Yaskawa INFORM job: u_tourne3TRJ4.JBI

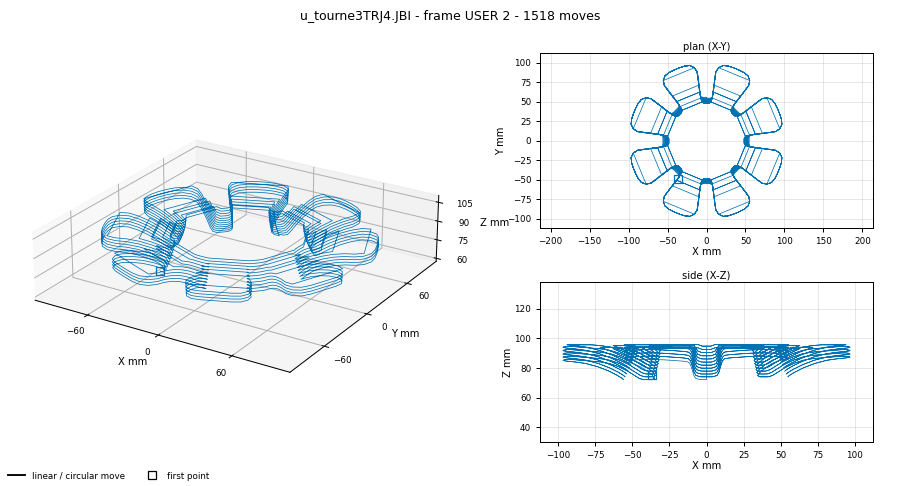
[picture p0: tool path of u_tourne3TRJ4.JBI in frame USER 2, 1518 of 1518 moves have a stored position in this frame; points joined in program order, loops and branches not executed]
/JOB
//NAME u_tourne3TRJ4
///FOLDERNAME DEMO
//POS
///NPOS 1518,0,1518,0,0,0
///USER 2
///TOOL 7
///POSTYPE USER
///RECTAN
///RCONF 1,0,0,0,0,0,0,0,0,0,0,0,0,0,0,0,0,0,0,0,0,0,0,0
C00000=-36.517,-48.718,75.143,177.9288,-0.0843,-14346.8537
C00001=-35.037,-45.351,73.015,-166.0442,10.7217,-14347.6887
C00002=-36.538,-42.505,72.166,-173.7278,29.8093,-14350.6829
C00003=-38.303,-40.803,72.129,179.7748,31.2094,-14353.1899
C00004=-39.567,-39.567,72.154,-180.0000,31.1989,-14355.0000
C00005=-40.803,-38.303,72.129,-179.7748,31.2094,-14356.8101
C00006=-42.506,-36.538,72.166,173.7274,29.8092,-14359.3178
C00007=-45.352,-35.037,73.015,166.0441,10.7215,-14362.3119
C00008=-48.718,-36.517,75.143,-177.9288,-0.0843,-14363.1463
C00009=-53.324,-40.007,78.036,-176.1608,-0.0420,-14363.1205
C00010=-59.196,-44.618,80.927,-175.6070,-0.0220,-14362.9934
C00011=-65.578,-49.604,83.062,-175.3163,-0.0261,-14362.8957
C00012=-71.524,-53.949,84.088,-175.5865,-0.7799,-14362.9735
C00013=-77.795,-55.184,84.621,-177.8577,-1.8362,-14364.6500
C00014=-83.601,-53.037,85.050,-179.4963,-1.2492,-14367.6087
C00015=-87.741,-47.957,85.481,179.9995,-0.0846,-14371.3401
C00016=-90.934,-41.602,85.762,-179.9996,-0.0128,-14375.4161
C00017=-93.717,-34.883,85.762,-179.9986,-0.0127,-14379.5839
C00018=-95.953,-28.131,85.481,179.9978,-0.0889,-14383.6602
C00019=-96.617,-21.612,85.050,179.4972,-1.2499,-14387.3912
C00020=-94.030,-15.989,84.621,177.8561,-1.8342,-14390.3496
C00021=-88.723,-12.427,84.088,175.5876,-0.7793,-14392.0267
C00022=-81.446,-11.295,83.062,175.3181,-0.0225,-14392.1045
C00023=-73.408,-10.308,80.927,175.6017,-0.0195,-14392.0068
C00024=-65.995,-9.417,78.036,176.1598,-0.0428,-14391.8791
C00025=-60.270,-8.627,75.143,177.9267,-0.0854,-14391.8541
C00026=-56.844,-7.293,73.015,-166.0480,10.7254,-14392.6890
C00027=-55.892,-4.219,72.166,-173.7293,29.8078,-14395.6832
C00028=-55.936,-1.768,72.129,179.7768,31.2086,-14398.1896
C00029=-55.957,0.000,72.154,-180.0000,31.1976,-14400.0000
C00030=-55.936,1.767,72.129,-179.7762,31.2086,-14401.8094
C00031=-55.892,4.220,72.166,173.7222,29.8074,-14404.3178
C00032=-56.844,7.293,73.015,166.0480,10.7254,-14407.3110
C00033=-60.270,8.627,75.143,-177.9267,-0.0854,-14408.1459
C00034=-65.995,9.417,78.036,-176.1598,-0.0428,-14408.1209
C00035=-73.408,10.308,80.927,-175.6017,-0.0195,-14407.9932
C00036=-81.446,11.295,83.062,-175.3181,-0.0225,-14407.8955
C00037=-88.723,12.427,84.088,-175.5876,-0.7793,-14407.9733
C00038=-94.030,15.989,84.621,-177.8561,-1.8342,-14409.6504
C00039=-96.617,21.612,85.050,-179.4972,-1.2499,-14412.6088
C00040=-95.953,28.131,85.481,-179.9978,-0.0889,-14416.3398
C00041=-93.717,34.883,85.762,179.9986,-0.0127,-14420.4161
C00042=-90.934,41.602,85.762,179.9996,-0.0128,-14424.5839
C00043=-87.741,47.957,85.481,-179.9995,-0.0846,-14428.6599
C00044=-83.601,53.037,85.050,179.4963,-1.2492,-14432.3913
C00045=-77.795,55.184,84.621,177.8577,-1.8362,-14435.3500
C00046=-71.524,53.949,84.088,175.5865,-0.7799,-14437.0265
C00047=-65.578,49.604,83.062,175.3163,-0.0261,-14437.1043
C00048=-59.196,44.618,80.927,175.6070,-0.0220,-14437.0066
C00049=-53.324,40.007,78.036,176.1608,-0.0420,-14436.8795
C00050=-48.718,36.517,75.143,177.9288,-0.0843,-14436.8537
C00051=-45.351,35.037,73.015,-166.0442,10.7217,-14437.6887
C00052=-42.505,36.538,72.166,-173.7278,29.8093,-14440.6829
C00053=-40.803,38.303,72.129,179.7748,31.2094,-14443.1899
C00054=-39.567,39.567,72.154,-180.0000,31.1989,-14445.0000
C00055=-38.303,40.803,72.129,-179.7748,31.2094,-14446.8101
C00056=-36.538,42.506,72.166,173.7274,29.8092,-14449.3178
C00057=-35.037,45.352,73.015,166.0441,10.7215,-14452.3119
C00058=-36.517,48.718,75.143,-177.9288,-0.0843,-14453.1463
C00059=-40.007,53.324,78.036,-176.1608,-0.0420,-14453.1205
C00060=-44.618,59.196,80.927,-175.6070,-0.0220,-14452.9934
C00061=-49.604,65.578,83.062,-175.3163,-0.0261,-14452.8957
C00062=-53.949,71.524,84.088,-175.5865,-0.7799,-14452.9735
C00063=-55.184,77.795,84.621,-177.8577,-1.8362,-14454.6500
C00064=-53.037,83.601,85.050,-179.4963,-1.2492,-14457.6087
C00065=-47.957,87.741,85.481,179.9995,-0.0846,-14461.3401
C00066=-41.602,90.934,85.762,-179.9996,-0.0128,-14465.4161
C00067=-34.883,93.717,85.762,-179.9986,-0.0127,-14469.5839
C00068=-28.131,95.953,85.481,179.9978,-0.0889,-14473.6602
C00069=-21.612,96.617,85.050,179.4972,-1.2499,-14477.3912
C00070=-15.989,94.030,84.621,177.8561,-1.8342,-14480.3496
C00071=-12.427,88.723,84.088,175.5876,-0.7793,-14482.0267
C00072=-11.295,81.446,83.062,175.3181,-0.0225,-14482.1045
C00073=-10.308,73.408,80.927,175.6017,-0.0195,-14482.0068
C00074=-9.417,65.995,78.036,176.1598,-0.0428,-14481.8791
C00075=-8.627,60.270,75.143,177.9267,-0.0854,-14481.8541
C00076=-7.293,56.844,73.015,-166.0480,10.7254,-14482.6890
C00077=-4.220,55.892,72.166,-173.7222,29.8074,-14485.6822
C00078=-1.767,55.936,72.129,179.7762,31.2086,-14488.1906
C00079=0.000,55.957,72.154,-180.0000,31.1976,-14490.0000
C00080=0.000,54.840,74.049,-180.0000,29.7413,-14490.0000
C00081=1.666,54.823,74.024,-179.8067,29.7500,-14491.7406
C00082=4.048,54.790,74.062,173.8586,28.2915,-14494.2255
C00083=7.088,55.804,74.943,167.0788,9.5543,-14497.2387
C00084=8.393,59.388,77.145,-177.8370,-0.0706,-14498.0440
C00085=9.180,65.335,80.122,-176.4294,-0.0310,-14497.9981
C00086=10.089,72.980,83.074,-176.0907,-0.0153,-14497.8709
C00087=11.094,81.206,85.240,-175.9759,-0.0117,-14497.7793
C00088=12.226,88.613,86.276,-176.2817,-0.6456,-14497.8555
C00089=15.808,94.009,86.813,-178.2035,-1.5233,-14499.5452
C00090=21.475,96.642,87.246,-179.5823,-1.0342,-14502.5282
C00091=28.048,95.980,87.679,179.9973,-0.0724,-14506.2898
C00092=34.856,93.728,87.962,179.9966,-0.0074,-14510.3994
C00093=41.629,90.922,87.962,179.9972,-0.0076,-14514.6009
C00094=48.035,87.701,87.679,-179.9999,-0.0718,-14518.7101
C00095=53.151,83.521,87.246,179.5838,-1.0323,-14522.4718
C00096=55.296,77.652,86.813,178.2066,-1.5235,-14525.4547
C00097=54.014,71.304,86.276,176.2804,-0.6460,-14527.1446
C00098=49.577,65.266,85.240,175.9790,-0.0155,-14527.2208
C00099=44.470,58.738,83.074,176.0895,-0.0120,-14527.1290
C00100=39.708,52.690,80.122,176.4261,-0.0301,-14527.0022
C00101=36.059,47.928,77.145,177.8373,-0.0709,-14526.9563
C00102=34.447,44.472,74.943,-167.0757,9.5522,-14527.7605
C00103=35.880,41.605,74.062,-173.8568,28.2919,-14530.7744
C00104=37.588,39.944,74.024,179.8046,29.7498,-14533.2595
C00105=38.778,38.778,74.049,-180.0000,29.7416,-14535.0000
C00106=39.943,37.588,74.024,-179.8042,29.7498,-14536.7398
C00107=41.605,35.880,74.062,173.8533,28.2853,-14539.2256
C00108=44.472,34.447,74.943,167.0757,9.5522,-14542.2395
C00109=47.928,36.059,77.145,-177.8373,-0.0709,-14543.0437
C00110=52.690,39.708,80.122,-176.4261,-0.0301,-14542.9978
C00111=58.738,44.470,83.074,-176.0895,-0.0120,-14542.8710
C00112=65.266,49.577,85.240,-175.9790,-0.0155,-14542.7792
C00113=71.304,54.014,86.276,-176.2804,-0.6460,-14542.8554
C00114=77.652,55.296,86.813,-178.2066,-1.5235,-14544.5453
C00115=83.521,53.151,87.246,-179.5838,-1.0323,-14547.5282
C00116=87.701,48.035,87.679,179.9999,-0.0718,-14551.2899
C00117=90.922,41.629,87.962,-179.9972,-0.0076,-14555.3991
C00118=93.728,34.856,87.962,-179.9966,-0.0074,-14559.6006
C00119=95.980,28.048,87.679,-179.9973,-0.0724,-14563.7102
C00120=96.642,21.475,87.246,179.5823,-1.0342,-14567.4718
C00121=94.009,15.808,86.813,178.2035,-1.5233,-14570.4548
C00122=88.613,12.226,86.276,176.2817,-0.6456,-14572.1445
C00123=81.206,11.094,85.240,175.9759,-0.0117,-14572.2207
C00124=72.980,10.089,83.074,176.0907,-0.0153,-14572.1291
C00125=65.335,9.180,80.122,176.4294,-0.0310,-14572.0019
C00126=59.388,8.393,77.145,177.8370,-0.0706,-14571.9560
C00127=55.804,7.088,74.943,-167.0788,9.5543,-14572.7613
C00128=54.790,4.048,74.062,-173.8586,28.2915,-14575.7745
C00129=54.823,1.666,74.024,179.8067,29.7500,-14578.2594
C00130=54.840,0.000,74.049,180.0000,29.7413,-14580.0000
C00131=54.823,-1.665,74.024,-179.8061,29.7500,-14581.7396
C00132=54.790,-4.048,74.062,173.8593,28.2888,-14584.2255
C00133=55.804,-7.088,74.943,167.0788,9.5543,-14587.2387
C00134=59.388,-8.393,77.145,-177.8370,-0.0706,-14588.0440
C00135=65.335,-9.180,80.122,-176.4294,-0.0310,-14587.9981
C00136=72.980,-10.089,83.074,-176.0907,-0.0153,-14587.8709
C00137=81.206,-11.094,85.240,-175.9759,-0.0117,-14587.7793
C00138=88.613,-12.226,86.276,-176.2817,-0.6456,-14587.8555
C00139=94.009,-15.808,86.813,-178.2035,-1.5233,-14589.5452
C00140=96.642,-21.475,87.246,-179.5823,-1.0342,-14592.5282
C00141=95.980,-28.048,87.679,179.9973,-0.0724,-14596.2898
C00142=93.728,-34.856,87.962,179.9966,-0.0074,-14600.3994
C00143=90.922,-41.629,87.962,179.9972,-0.0076,-14604.6009
C00144=87.701,-48.035,87.679,-179.9999,-0.0718,-14608.7101
C00145=83.521,-53.151,87.246,179.5838,-1.0323,-14612.4718
C00146=77.652,-55.296,86.813,178.2066,-1.5235,-14615.4547
C00147=71.304,-54.014,86.276,176.2804,-0.6460,-14617.1446
C00148=65.266,-49.577,85.240,175.9790,-0.0155,-14617.2208
C00149=58.738,-44.470,83.074,176.0895,-0.0120,-14617.1290
C00150=52.690,-39.708,80.122,176.4261,-0.0301,-14617.0022
C00151=47.928,-36.059,77.145,177.8373,-0.0709,-14616.9563
C00152=44.472,-34.447,74.943,-167.0757,9.5522,-14617.7605
C00153=41.605,-35.880,74.062,-173.8568,28.2919,-14620.7744
C00154=39.944,-37.588,74.024,179.8046,29.7498,-14623.2595
C00155=38.778,-38.778,74.049,180.0000,29.7416,-14625.0000
C00156=37.588,-39.943,74.024,-179.8042,29.7498,-14626.7398
C00157=35.880,-41.605,74.062,173.8533,28.2853,-14629.2256
C00158=34.447,-44.472,74.943,167.0757,9.5522,-14632.2395
C00159=36.059,-47.928,77.145,-177.8373,-0.0709,-14633.0437
C00160=39.708,-52.690,80.122,-176.4261,-0.0301,-14632.9978
C00161=44.470,-58.738,83.074,-176.0895,-0.0120,-14632.8710
C00162=49.577,-65.266,85.240,-175.9790,-0.0155,-14632.7792
C00163=54.014,-71.304,86.276,-176.2804,-0.6460,-14632.8554
C00164=55.296,-77.652,86.813,-178.2066,-1.5235,-14634.5453
C00165=53.151,-83.521,87.246,-179.5838,-1.0323,-14637.5282
C00166=48.035,-87.701,87.679,179.9999,-0.0718,-14641.2899
C00167=41.629,-90.922,87.962,-179.9972,-0.0076,-14645.3991
C00168=34.856,-93.728,87.962,-179.9966,-0.0074,-14649.6006
C00169=28.048,-95.980,87.679,-179.9973,-0.0724,-14653.7102
C00170=21.475,-96.642,87.246,179.5823,-1.0342,-14657.4718
C00171=15.808,-94.009,86.813,178.2035,-1.5233,-14660.4548
C00172=12.226,-88.613,86.276,176.2817,-0.6456,-14662.1445
C00173=11.094,-81.206,85.240,175.9759,-0.0117,-14662.2207
C00174=10.089,-72.980,83.074,176.0907,-0.0153,-14662.1291
C00175=9.180,-65.335,80.122,176.4294,-0.0310,-14662.0019
C00176=8.393,-59.388,77.145,177.8370,-0.0706,-14661.9560
C00177=7.088,-55.804,74.943,-167.0788,9.5543,-14662.7613
C00178=4.048,-54.790,74.062,-173.8586,28.2915,-14665.7745
C00179=1.666,-54.823,74.024,179.8067,29.7500,-14668.2594
C00180=0.000,-54.840,74.049,-180.0000,29.7413,-14670.0000
C00181=0.000,-54.840,74.049,-180.0000,29.7413,-14670.0000
C00182=-1.665,-54.823,74.024,-179.8061,29.7500,-14671.7396
C00183=-4.048,-54.790,74.062,173.8593,28.2888,-14674.2255
C00184=-7.088,-55.804,74.943,167.0788,9.5543,-14677.2387
C00185=-8.393,-59.388,77.145,-177.8370,-0.0706,-14678.0440
C00186=-9.180,-65.335,80.122,-176.4294,-0.0310,-14677.9981
C00187=-10.089,-72.980,83.074,-176.0907,-0.0153,-14677.8709
C00188=-11.094,-81.206,85.240,-175.9759,-0.0117,-14677.7793
C00189=-12.226,-88.613,86.276,-176.2817,-0.6456,-14677.8555
C00190=-15.808,-94.009,86.813,-178.2035,-1.5233,-14679.5452
C00191=-21.475,-96.642,87.246,-179.5823,-1.0342,-14682.5282
C00192=-28.048,-95.980,87.679,179.9973,-0.0724,-14686.2898
C00193=-34.856,-93.728,87.962,179.9966,-0.0074,-14690.3994
C00194=-41.629,-90.922,87.962,179.9972,-0.0076,-14694.6009
C00195=-48.035,-87.701,87.679,-179.9999,-0.0718,-14698.7101
C00196=-53.151,-83.521,87.246,179.5838,-1.0323,-14702.4718
C00197=-55.296,-77.652,86.813,178.2066,-1.5235,-14705.4547
C00198=-54.014,-71.304,86.276,176.2804,-0.6460,-14707.1446
C00199=-49.577,-65.266,85.240,175.9790,-0.0155,-14707.2208
C00200=-44.470,-58.738,83.074,176.0895,-0.0120,-14707.1290
C00201=-39.708,-52.690,80.122,176.4261,-0.0301,-14707.0022
C00202=-36.059,-47.928,77.145,177.8373,-0.0709,-14706.9563
C00203=-34.447,-44.472,74.943,-167.0757,9.5522,-14707.7605
C00204=-35.880,-41.605,74.062,-173.8568,28.2919,-14710.7744
C00205=-37.588,-39.944,74.024,179.8046,29.7498,-14713.2595
C00206=-38.778,-38.778,74.049,-180.0000,29.7416,-14715.0000
C00207=-39.943,-37.588,74.024,-179.8042,29.7498,-14716.7398
C00208=-41.605,-35.880,74.062,173.8533,28.2853,-14719.2256
C00209=-44.472,-34.447,74.943,167.0757,9.5522,-14722.2395
C00210=-47.928,-36.059,77.145,-177.8373,-0.0709,-14723.0437
C00211=-52.690,-39.708,80.122,-176.4261,-0.0301,-14722.9978
C00212=-58.738,-44.470,83.074,-176.0895,-0.0120,-14722.8710
C00213=-65.266,-49.577,85.240,-175.9790,-0.0155,-14722.7792
C00214=-71.304,-54.014,86.276,-176.2804,-0.6460,-14722.8554
C00215=-77.652,-55.296,86.813,-178.2066,-1.5235,-14724.5453
C00216=-83.521,-53.151,87.246,-179.5838,-1.0323,-14727.5282
C00217=-87.701,-48.035,87.679,179.9999,-0.0718,-14731.2899
C00218=-90.922,-41.629,87.962,-179.9972,-0.0076,-14735.3991
C00219=-93.728,-34.856,87.962,-179.9966,-0.0074,-14739.6006
C00220=-95.980,-28.048,87.679,-179.9973,-0.0724,-14743.7102
C00221=-96.642,-21.475,87.246,179.5823,-1.0342,-14747.4718
C00222=-94.009,-15.808,86.813,178.2035,-1.5233,-14750.4548
C00223=-88.613,-12.226,86.276,176.2817,-0.6456,-14752.1445
C00224=-81.206,-11.094,85.240,175.9759,-0.0117,-14752.2207
C00225=-72.980,-10.089,83.074,176.0907,-0.0153,-14752.1291
C00226=-65.335,-9.180,80.122,176.4294,-0.0310,-14752.0019
C00227=-59.388,-8.393,77.145,177.8370,-0.0706,-14751.9560
C00228=-55.804,-7.088,74.943,-167.0788,9.5543,-14752.7613
C00229=-54.790,-4.048,74.062,-173.8586,28.2915,-14755.7745
C00230=-54.823,-1.666,74.024,179.8067,29.7500,-14758.2594
C00231=-54.840,0.000,74.049,-180.0000,29.7413,-14760.0000
C00232=-54.823,1.665,74.024,-179.8061,29.7500,-14761.7396
C00233=-54.790,4.048,74.062,173.8593,28.2888,-14764.2255
C00234=-55.804,7.088,74.943,167.0788,9.5543,-14767.2387
C00235=-59.388,8.393,77.145,-177.8370,-0.0706,-14768.0440
C00236=-65.335,9.180,80.122,-176.4294,-0.0310,-14767.9981
C00237=-72.980,10.089,83.074,-176.0907,-0.0153,-14767.8709
C00238=-81.206,11.094,85.240,-175.9759,-0.0117,-14767.7793
C00239=-88.613,12.226,86.276,-176.2817,-0.6456,-14767.8555
C00240=-94.009,15.808,86.813,-178.2035,-1.5233,-14769.5452
C00241=-96.642,21.475,87.246,-179.5823,-1.0342,-14772.5282
C00242=-95.980,28.048,87.679,179.9973,-0.0724,-14776.2898
C00243=-93.728,34.856,87.962,179.9966,-0.0074,-14780.3994
C00244=-90.922,41.629,87.962,179.9972,-0.0076,-14784.6009
C00245=-87.701,48.035,87.679,-179.9999,-0.0718,-14788.7101
C00246=-83.521,53.151,87.246,179.5838,-1.0323,-14792.4718
C00247=-77.652,55.296,86.813,178.2066,-1.5235,-14795.4547
C00248=-71.304,54.014,86.276,176.2804,-0.6460,-14797.1446
C00249=-65.266,49.577,85.240,175.9790,-0.0155,-14797.2208
C00250=-58.738,44.470,83.074,176.0895,-0.0120,-14797.1290
C00251=-52.690,39.708,80.122,176.4261,-0.0301,-14797.0022
C00252=-47.928,36.059,77.145,177.8373,-0.0709,-14796.9563
C00253=-44.472,34.447,74.943,-167.0757,9.5522,-14797.7605
C00254=-41.605,35.880,74.062,-173.8568,28.2919,-14800.7744
C00255=-39.944,37.588,74.024,179.8046,29.7498,-14803.2595
C00256=-38.778,38.778,74.049,-180.0000,29.7416,-14805.0000
C00257=-37.588,39.943,74.024,-179.8042,29.7498,-14806.7398
C00258=-35.880,41.605,74.062,173.8533,28.2853,-14809.2256
C00259=-34.447,44.472,74.943,167.0757,9.5522,-14812.2395
C00260=-36.059,47.928,77.145,-177.8373,-0.0709,-14813.0437
C00261=-39.708,52.690,80.122,-176.4261,-0.0301,-14812.9978
C00262=-44.470,58.738,83.074,-176.0895,-0.0120,-14812.8710
C00263=-49.577,65.266,85.240,-175.9790,-0.0155,-14812.7792
C00264=-54.014,71.304,86.276,-176.2804,-0.6460,-14812.8554
C00265=-55.296,77.652,86.813,-178.2066,-1.5235,-14814.5453
C00266=-53.151,83.521,87.246,-179.5838,-1.0323,-14817.5282
C00267=-48.035,87.701,87.679,179.9999,-0.0718,-14821.2899
C00268=-41.629,90.922,87.962,-179.9972,-0.0076,-14825.3991
C00269=-34.856,93.728,87.962,-179.9966,-0.0074,-14829.6006
C00270=-28.048,95.980,87.679,-179.9973,-0.0724,-14833.7102
C00271=-21.475,96.642,87.246,179.5823,-1.0342,-14837.4718
C00272=-15.808,94.009,86.813,178.2035,-1.5233,-14840.4548
C00273=-12.226,88.613,86.276,176.2817,-0.6456,-14842.1445
C00274=-11.094,81.206,85.240,175.9759,-0.0117,-14842.2207
C00275=-10.089,72.980,83.074,176.0907,-0.0153,-14842.1291
C00276=-9.180,65.335,80.122,176.4294,-0.0310,-14842.0019
C00277=-8.393,59.388,77.145,177.8370,-0.0706,-14841.9560
C00278=-7.088,55.804,74.943,-167.0788,9.5543,-14842.7613
C00279=-4.048,54.790,74.062,-173.8593,28.2888,-14845.7745
C00280=-1.665,54.823,74.024,179.8061,29.7500,-14848.2604
C00281=0.000,54.840,74.049,180.0000,29.7413,-14850.0000
C00282=0.000,53.776,75.975,180.0000,28.1001,-14850.0000
C00283=1.568,53.762,75.948,-179.8334,28.1117,-14851.6706
C00284=3.884,53.739,75.988,174.0567,26.6026,-14854.1339
C00285=6.894,54.818,76.900,168.1623,8.4382,-14857.1680
C00286=8.175,58.565,79.173,-177.8225,-0.0548,-14857.9465
C00287=8.965,64.737,82.228,-176.7507,-0.0188,-14857.8844
C00288=9.898,72.606,85.234,-176.6314,-0.0094,-14857.7630
C00289=10.924,81.005,87.424,-176.6961,-0.0057,-14857.6803
C00290=12.061,88.524,88.468,-177.0328,-0.5045,-14857.7585
C00291=15.662,93.991,89.008,-178.5867,-1.1939,-14859.4604
C00292=21.365,96.662,89.443,-179.6771,-0.7971,-14862.4636
C00293=27.983,96.002,89.878,179.9979,-0.0543,-14866.2505
C00294=34.834,93.736,90.162,-179.9980,-0.0054,-14870.3860
C00295=41.650,90.913,90.162,-179.9976,-0.0052,-14874.6140
C00296=48.097,87.670,89.878,179.9969,-0.0540,-14878.7498
C00297=53.243,83.458,89.443,179.6739,-0.7993,-14882.5363
C00298=55.387,77.537,89.008,178.5849,-1.1940,-14885.5394
C00299=54.067,71.124,88.468,177.0304,-0.5081,-14887.2413
C00300=49.554,65.004,87.424,176.6978,-0.0087,-14887.3191
C00301=44.341,58.339,85.234,176.6315,-0.0113,-14887.2369
C00302=39.437,52.115,82.228,176.7520,-0.0208,-14887.1159
C00303=35.631,47.192,79.173,177.8236,-0.0563,-14887.0536
C00304=33.888,43.637,76.900,-168.1624,8.4405,-14887.8325
C00305=35.253,40.746,75.988,-174.0559,26.5997,-14890.8660
C00306=36.906,39.124,75.948,179.8313,28.1098,-14893.3290
C00307=38.025,38.025,75.975,-180.0000,28.0967,-14895.0000
C00308=39.124,36.906,75.948,-179.8313,28.1098,-14896.6710
C00309=40.746,35.253,75.988,174.0559,26.5997,-14899.1340
C00310=43.637,33.888,76.901,168.1624,8.4405,-14902.1675
C00311=47.192,35.631,79.173,-177.8236,-0.0563,-14902.9464
C00312=52.115,39.437,82.228,-176.7520,-0.0208,-14902.8841
C00313=58.339,44.341,85.234,-176.6315,-0.0113,-14902.7631
C00314=65.004,49.554,87.424,-176.6978,-0.0087,-14902.6809
C00315=71.124,54.067,88.468,-177.0304,-0.5081,-14902.7587
C00316=77.537,55.387,89.008,-178.5849,-1.1940,-14904.4606
C00317=83.458,53.243,89.443,-179.6739,-0.7993,-14907.4637
C00318=87.670,48.097,89.878,-179.9969,-0.0540,-14911.2502
C00319=90.913,41.650,90.162,179.9976,-0.0052,-14915.3860
C00320=93.736,34.834,90.162,179.9980,-0.0054,-14919.6140
C00321=96.002,27.983,89.878,-179.9979,-0.0543,-14923.7495
C00322=96.662,21.365,89.443,179.6771,-0.7971,-14927.5364
C00323=93.991,15.662,89.008,178.5867,-1.1939,-14930.5396
C00324=88.524,12.061,88.468,177.0328,-0.5045,-14932.2415
C00325=81.005,10.924,87.424,176.6961,-0.0057,-14932.3197
C00326=72.606,9.898,85.234,176.6314,-0.0094,-14932.2370
C00327=64.737,8.965,82.228,176.7507,-0.0188,-14932.1156
C00328=58.565,8.175,79.173,177.8225,-0.0548,-14932.0535
C00329=54.818,6.894,76.900,-168.1623,8.4382,-14932.8320
C00330=53.739,3.884,75.988,-174.0567,26.6026,-14935.8661
C00331=53.762,1.568,75.948,179.8334,28.1117,-14938.3294
C00332=53.776,0.000,75.975,180.0000,28.1001,-14940.0000
C00333=53.762,-1.568,75.948,-179.8334,28.1117,-14941.6706
C00334=53.739,-3.885,75.988,174.0562,26.6025,-14944.1349
C00335=54.819,-6.894,76.901,168.1623,8.4383,-14947.1678
C00336=58.565,-8.175,79.173,-177.8225,-0.0548,-14947.9465
C00337=64.737,-8.965,82.228,-176.7507,-0.0188,-14947.8844
C00338=72.606,-9.898,85.234,-176.6314,-0.0094,-14947.7630
C00339=81.005,-10.924,87.424,-176.6961,-0.0057,-14947.6803
C00340=88.524,-12.061,88.468,-177.0328,-0.5045,-14947.7585
C00341=93.991,-15.662,89.008,-178.5867,-1.1939,-14949.4604
C00342=96.662,-21.365,89.443,-179.6771,-0.7971,-14952.4636
C00343=96.002,-27.983,89.878,179.9979,-0.0543,-14956.2505
C00344=93.736,-34.834,90.162,-179.9980,-0.0054,-14960.3860
C00345=90.913,-41.650,90.162,-179.9976,-0.0052,-14964.6140
C00346=87.670,-48.097,89.878,179.9969,-0.0540,-14968.7498
C00347=83.458,-53.243,89.443,179.6739,-0.7993,-14972.5363
C00348=77.537,-55.387,89.008,178.5849,-1.1940,-14975.5394
C00349=71.124,-54.067,88.468,177.0304,-0.5081,-14977.2413
C00350=65.004,-49.554,87.424,176.6978,-0.0087,-14977.3191
C00351=58.339,-44.341,85.234,176.6315,-0.0113,-14977.2369
C00352=52.115,-39.437,82.228,176.7520,-0.0208,-14977.1159
C00353=47.192,-35.631,79.173,177.8236,-0.0563,-14977.0536
C00354=43.637,-33.888,76.900,-168.1624,8.4405,-14977.8325
C00355=40.746,-35.253,75.988,-174.0559,26.5997,-14980.8660
C00356=39.124,-36.906,75.948,179.8313,28.1098,-14983.3290
C00357=38.025,-38.025,75.975,-180.0000,28.0967,-14985.0000
C00358=36.906,-39.124,75.948,-179.8313,28.1098,-14986.6710
C00359=35.253,-40.746,75.988,174.0559,26.5997,-14989.1340
C00360=33.888,-43.637,76.901,168.1624,8.4405,-14992.1675
C00361=35.631,-47.192,79.173,-177.8236,-0.0563,-14992.9464
C00362=39.437,-52.115,82.228,-176.7520,-0.0208,-14992.8841
C00363=44.341,-58.339,85.234,-176.6315,-0.0113,-14992.7631
C00364=49.554,-65.004,87.424,-176.6978,-0.0087,-14992.6809
C00365=54.067,-71.124,88.468,-177.0304,-0.5081,-14992.7587
C00366=55.387,-77.537,89.008,-178.5849,-1.1940,-14994.4606
C00367=53.243,-83.458,89.443,-179.6739,-0.7993,-14997.4637
C00368=48.097,-87.670,89.878,-179.9969,-0.0540,-15001.2502
C00369=41.650,-90.913,90.162,179.9976,-0.0052,-15005.3860
C00370=34.834,-93.736,90.162,179.9980,-0.0054,-15009.6140
C00371=27.983,-96.002,89.878,-179.9979,-0.0543,-15013.7495
C00372=21.365,-96.662,89.443,179.6771,-0.7971,-15017.5364
C00373=15.662,-93.991,89.008,178.5867,-1.1939,-15020.5396
C00374=12.061,-88.524,88.468,177.0328,-0.5045,-15022.2415
C00375=10.924,-81.005,87.424,176.6961,-0.0057,-15022.3197
C00376=9.898,-72.606,85.234,176.6314,-0.0094,-15022.2370
C00377=8.965,-64.737,82.228,176.7507,-0.0188,-15022.1156
C00378=8.175,-58.565,79.173,177.8225,-0.0548,-15022.0535
C00379=6.894,-54.818,76.900,-168.1623,8.4382,-15022.8320
C00380=3.884,-53.739,75.988,-174.0567,26.6026,-15025.8661
C00381=1.568,-53.762,75.948,179.8334,28.1117,-15028.3294
C00382=0.000,-53.776,75.975,180.0000,28.1001,-15030.0000
C00383=0.000,-53.776,75.975,180.0000,28.1001,-15030.0000
C00384=-1.568,-53.762,75.948,-179.8334,28.1117,-15031.6706
C00385=-3.885,-53.739,75.988,174.0562,26.6025,-15034.1349
C00386=-6.894,-54.819,76.901,168.1623,8.4383,-15037.1678
C00387=-8.175,-58.565,79.173,-177.8225,-0.0548,-15037.9465
C00388=-8.965,-64.737,82.228,-176.7507,-0.0188,-15037.8844
C00389=-9.898,-72.606,85.234,-176.6314,-0.0094,-15037.7630
C00390=-10.924,-81.005,87.424,-176.6961,-0.0057,-15037.6803
C00391=-12.061,-88.524,88.468,-177.0328,-0.5045,-15037.7585
C00392=-15.662,-93.991,89.008,-178.5867,-1.1939,-15039.4604
C00393=-21.365,-96.662,89.443,-179.6771,-0.7971,-15042.4636
C00394=-27.983,-96.002,89.878,179.9979,-0.0543,-15046.2505
C00395=-34.834,-93.736,90.162,-179.9980,-0.0054,-15050.3860
C00396=-41.650,-90.913,90.162,-179.9976,-0.0052,-15054.6140
C00397=-48.097,-87.670,89.878,179.9969,-0.0540,-15058.7498
C00398=-53.243,-83.458,89.443,179.6739,-0.7993,-15062.5363
C00399=-55.387,-77.537,89.008,178.5849,-1.1940,-15065.5394
C00400=-54.067,-71.124,88.468,177.0304,-0.5081,-15067.2413
C00401=-49.554,-65.004,87.424,176.6978,-0.0087,-15067.3191
C00402=-44.341,-58.339,85.234,176.6315,-0.0113,-15067.2369
C00403=-39.437,-52.115,82.228,176.7520,-0.0208,-15067.1159
C00404=-35.631,-47.192,79.173,177.8236,-0.0563,-15067.0536
C00405=-33.888,-43.637,76.900,-168.1624,8.4405,-15067.8325
C00406=-35.253,-40.746,75.988,-174.0559,26.5997,-15070.8660
C00407=-36.906,-39.124,75.948,179.8313,28.1098,-15073.3290
C00408=-38.025,-38.025,75.975,-180.0000,28.0967,-15075.0000
C00409=-39.124,-36.906,75.948,-179.8313,28.1098,-15076.6710
C00410=-40.746,-35.253,75.988,174.0559,26.5997,-15079.1340
C00411=-43.637,-33.888,76.901,168.1624,8.4405,-15082.1675
C00412=-47.192,-35.631,79.173,-177.8236,-0.0563,-15082.9464
C00413=-52.115,-39.437,82.228,-176.7520,-0.0208,-15082.8841
C00414=-58.339,-44.341,85.234,-176.6315,-0.0113,-15082.7631
C00415=-65.004,-49.554,87.424,-176.6978,-0.0087,-15082.6809
C00416=-71.124,-54.067,88.468,-177.0304,-0.5081,-15082.7587
C00417=-77.537,-55.387,89.008,-178.5849,-1.1940,-15084.4606
C00418=-83.458,-53.243,89.443,-179.6739,-0.7993,-15087.4637
C00419=-87.670,-48.097,89.878,-179.9969,-0.0540,-15091.2502
C00420=-90.913,-41.650,90.162,179.9976,-0.0052,-15095.3860
C00421=-93.736,-34.834,90.162,179.9980,-0.0054,-15099.6140
C00422=-96.002,-27.983,89.878,-179.9979,-0.0543,-15103.7495
C00423=-96.662,-21.365,89.443,179.6771,-0.7971,-15107.5364
C00424=-93.991,-15.662,89.008,178.5867,-1.1939,-15110.5396
C00425=-88.524,-12.061,88.468,177.0328,-0.5045,-15112.2415
C00426=-81.005,-10.924,87.424,176.6961,-0.0057,-15112.3197
C00427=-72.606,-9.898,85.234,176.6314,-0.0094,-15112.2370
C00428=-64.737,-8.965,82.228,176.7507,-0.0188,-15112.1156
C00429=-58.565,-8.175,79.173,177.8225,-0.0548,-15112.0535
C00430=-54.818,-6.894,76.900,-168.1623,8.4382,-15112.8320
C00431=-53.739,-3.884,75.988,-174.0567,26.6026,-15115.8661
C00432=-53.762,-1.568,75.948,179.8334,28.1117,-15118.3294
C00433=-53.776,0.000,75.975,180.0000,28.1001,-15120.0000
C00434=-53.762,1.568,75.948,-179.8334,28.1117,-15121.6706
C00435=-53.739,3.885,75.988,174.0562,26.6025,-15124.1349
C00436=-54.819,6.894,76.901,168.1623,8.4383,-15127.1678
C00437=-58.565,8.175,79.173,-177.8225,-0.0548,-15127.9465
C00438=-64.737,8.965,82.228,-176.7507,-0.0188,-15127.8844
C00439=-72.606,9.898,85.234,-176.6314,-0.0094,-15127.7630
C00440=-81.005,10.924,87.424,-176.6961,-0.0057,-15127.6803
C00441=-88.524,12.061,88.468,-177.0328,-0.5045,-15127.7585
C00442=-93.991,15.662,89.008,-178.5867,-1.1939,-15129.4604
C00443=-96.662,21.365,89.443,-179.6771,-0.7971,-15132.4636
C00444=-96.002,27.983,89.878,179.9979,-0.0543,-15136.2505
C00445=-93.736,34.834,90.162,-179.9980,-0.0054,-15140.3860
C00446=-90.913,41.650,90.162,-179.9976,-0.0052,-15144.6140
C00447=-87.670,48.097,89.878,179.9969,-0.0540,-15148.7498
C00448=-83.458,53.243,89.443,179.6739,-0.7993,-15152.5363
C00449=-77.537,55.387,89.008,178.5849,-1.1940,-15155.5394
C00450=-71.124,54.067,88.468,177.0304,-0.5081,-15157.2413
C00451=-65.004,49.554,87.424,176.6978,-0.0087,-15157.3191
C00452=-58.339,44.341,85.234,176.6315,-0.0113,-15157.2369
C00453=-52.115,39.437,82.228,176.7520,-0.0208,-15157.1159
C00454=-47.192,35.631,79.173,177.8236,-0.0563,-15157.0536
C00455=-43.637,33.888,76.900,-168.1624,8.4405,-15157.8325
C00456=-40.746,35.253,75.988,-174.0559,26.5997,-15160.8660
C00457=-39.124,36.906,75.948,179.8313,28.1098,-15163.3290
C00458=-38.025,38.025,75.975,-180.0000,28.0967,-15165.0000
C00459=-36.906,39.124,75.948,-179.8313,28.1098,-15166.6710
C00460=-35.253,40.746,75.988,174.0559,26.5997,-15169.1340
C00461=-33.888,43.637,76.901,168.1624,8.4405,-15172.1675
C00462=-35.631,47.192,79.173,-177.8236,-0.0563,-15172.9464
C00463=-39.437,52.115,82.228,-176.7520,-0.0208,-15172.8841
C00464=-44.341,58.339,85.234,-176.6315,-0.0113,-15172.7631
C00465=-49.554,65.004,87.424,-176.6978,-0.0087,-15172.6809
C00466=-54.067,71.124,88.468,-177.0304,-0.5081,-15172.7587
C00467=-55.387,77.537,89.008,-178.5849,-1.1940,-15174.4606
C00468=-53.243,83.458,89.443,-179.6739,-0.7993,-15177.4637
C00469=-48.097,87.670,89.878,-179.9969,-0.0540,-15181.2502
C00470=-41.650,90.913,90.162,179.9976,-0.0052,-15185.3860
C00471=-34.834,93.736,90.162,179.9980,-0.0054,-15189.6140
C00472=-27.983,96.002,89.878,-179.9979,-0.0543,-15193.7495
C00473=-21.365,96.662,89.443,179.6771,-0.7971,-15197.5364
C00474=-15.662,93.991,89.008,178.5867,-1.1939,-15200.5396
C00475=-12.061,88.524,88.468,177.0328,-0.5045,-15202.2415
C00476=-10.924,81.005,87.424,176.6961,-0.0057,-15202.3197
C00477=-9.898,72.606,85.234,176.6314,-0.0094,-15202.2370
C00478=-8.965,64.737,82.228,176.7507,-0.0188,-15202.1156
C00479=-8.175,58.565,79.173,177.8225,-0.0548,-15202.0535
C00480=-6.894,54.819,76.901,-168.1623,8.4383,-15202.8322
C00481=-3.885,53.739,75.988,-174.0562,26.6025,-15205.8651
C00482=-1.568,53.762,75.948,179.8334,28.1117,-15208.3294
C00483=0.000,53.776,75.975,-180.0000,28.1001,-15210.0000
C00484=0.000,52.771,77.932,-180.0000,26.2576,-15210.0000
C00485=1.476,52.759,77.904,-179.8644,26.2720,-15211.6025
C00486=3.730,52.747,77.945,174.3297,24.7331,-15214.0449
C00487=6.711,53.894,78.888,169.2924,7.3770,-15217.0981
C00488=7.974,57.808,81.229,-177.8824,-0.0435,-15217.8538
C00489=8.774,64.206,84.354,-177.1343,-0.0134,-15217.7815
C00490=9.737,72.291,87.405,-177.2235,-0.0020,-15217.6711
C00491=10.790,80.844,89.614,-177.4669,-0.0031,-15217.6022
C00492=11.935,88.455,90.663,-177.8347,-0.3615,-15217.6844
C00493=15.553,93.978,91.206,-179.0014,-0.8397,-15219.3971
C00494=21.285,96.677,91.642,-179.7804,-0.5442,-15222.4165
C00495=27.936,96.017,92.077,179.9986,-0.0362,-15226.2223
C00496=34.820,93.742,92.362,-179.9980,-0.0054,-15230.3773
C00497=41.664,90.907,92.362,-179.9976,-0.0052,-15234.6227
C00498=48.140,87.648,92.077,-179.9985,-0.0384,-15238.7775
C00499=53.310,83.412,91.642,179.7765,-0.5441,-15242.5833
C00500=55.455,77.451,91.206,179.0023,-0.8412,-15245.6027
C00501=54.108,70.986,90.663,177.8365,-0.3666,-15247.3159
C00502=49.536,64.795,89.614,177.4688,-0.0016,-15247.3980
C00503=44.233,58.003,87.405,177.2268,-0.0027,-15247.3291
C00504=39.197,51.604,84.354,177.1305,-0.0129,-15247.2193
C00505=35.238,46.514,81.229,177.8797,-0.0389,-15247.1468
C00506=33.363,42.854,78.888,-169.2963,7.3773,-15247.9017
C00507=34.660,39.935,77.945,-174.3268,24.7330,-15250.9551
C00508=36.262,38.350,77.904,179.8603,26.2704,-15253.3970
C00509=37.314,37.314,77.932,-180.0000,26.2558,-15255.0000
C00510=38.350,36.262,77.904,-179.8603,26.2704,-15256.6030
C00511=39.935,34.660,77.945,174.3268,24.7330,-15259.0449
C00512=42.854,33.363,78.888,169.2928,7.3727,-15262.0983
C00513=46.514,35.238,81.229,-177.8797,-0.0389,-15262.8532
C00514=51.604,39.197,84.354,-177.1305,-0.0129,-15262.7807
C00515=58.003,44.233,87.405,-177.2268,-0.0027,-15262.6709
C00516=64.795,49.536,89.614,-177.4688,-0.0016,-15262.6020
C00517=70.986,54.108,90.663,-177.8365,-0.3666,-15262.6841
C00518=77.451,55.455,91.206,-179.0023,-0.8412,-15264.3973
C00519=83.412,53.310,91.642,-179.7765,-0.5441,-15267.4167
C00520=87.648,48.140,92.077,179.9985,-0.0384,-15271.2225
C00521=90.907,41.664,92.362,179.9976,-0.0052,-15275.3773
C00522=93.742,34.820,92.362,179.9980,-0.0054,-15279.6227
C00523=96.017,27.936,92.077,-179.9986,-0.0362,-15283.7777
C00524=96.677,21.285,91.642,179.7804,-0.5442,-15287.5835
C00525=93.978,15.553,91.206,179.0014,-0.8397,-15290.6029
C00526=88.455,11.935,90.663,177.8347,-0.3615,-15292.3156
C00527=80.844,10.790,89.614,177.4669,-0.0031,-15292.3978
C00528=72.291,9.737,87.405,177.2235,-0.0020,-15292.3289
C00529=64.206,8.774,84.354,177.1343,-0.0134,-15292.2185
C00530=57.808,7.974,81.229,177.8824,-0.0435,-15292.1462
C00531=53.894,6.711,78.888,-169.2924,7.3770,-15292.9019
C00532=52.747,3.730,77.945,-174.3297,24.7331,-15295.9551
C00533=52.759,1.476,77.904,179.8644,26.2720,-15298.3975
C00534=52.771,0.000,77.932,-180.0000,26.2576,-15300.0000
C00535=52.759,-1.476,77.904,-179.8644,26.2720,-15301.6025
C00536=52.747,-3.730,77.945,174.3235,24.7327,-15304.0449
C00537=53.894,-6.711,78.888,169.2924,7.3770,-15307.0981
C00538=57.808,-7.974,81.229,-177.8824,-0.0435,-15307.8538
C00539=64.206,-8.774,84.354,-177.1343,-0.0134,-15307.7815
C00540=72.291,-9.737,87.405,-177.2235,-0.0020,-15307.6711
C00541=80.844,-10.790,89.614,-177.4669,-0.0031,-15307.6022
C00542=88.455,-11.935,90.663,-177.8347,-0.3615,-15307.6844
C00543=93.978,-15.553,91.206,-179.0014,-0.8397,-15309.3971
C00544=96.677,-21.285,91.642,-179.7804,-0.5442,-15312.4165
C00545=96.017,-27.936,92.077,179.9986,-0.0362,-15316.2223
C00546=93.742,-34.820,92.362,-179.9980,-0.0054,-15320.3773
C00547=90.907,-41.664,92.362,-179.9976,-0.0052,-15324.6227
C00548=87.648,-48.140,92.077,-179.9985,-0.0384,-15328.7775
C00549=83.412,-53.310,91.642,179.7765,-0.5441,-15332.5833
C00550=77.451,-55.455,91.206,179.0023,-0.8412,-15335.6027
C00551=70.986,-54.108,90.663,177.8365,-0.3666,-15337.3159
C00552=64.795,-49.536,89.614,177.4688,-0.0016,-15337.3980
C00553=58.003,-44.233,87.405,177.2268,-0.0027,-15337.3291
C00554=51.604,-39.197,84.354,177.1305,-0.0129,-15337.2193
C00555=46.514,-35.238,81.229,177.8797,-0.0389,-15337.1468
C00556=42.854,-33.363,78.888,-169.2963,7.3773,-15337.9017
C00557=39.935,-34.660,77.945,-174.3268,24.7330,-15340.9551
C00558=38.350,-36.262,77.904,179.8603,26.2704,-15343.3970
C00559=37.314,-37.314,77.932,180.0000,26.2558,-15345.0000
C00560=36.262,-38.350,77.904,-179.8603,26.2704,-15346.6030
C00561=34.660,-39.935,77.945,174.3268,24.7330,-15349.0449
C00562=33.363,-42.854,78.888,169.2928,7.3727,-15352.0983
C00563=35.238,-46.514,81.229,-177.8797,-0.0389,-15352.8532
C00564=39.197,-51.604,84.354,-177.1305,-0.0129,-15352.7807
C00565=44.233,-58.003,87.405,-177.2268,-0.0027,-15352.6709
C00566=49.536,-64.795,89.614,-177.4688,-0.0016,-15352.6020
C00567=54.108,-70.986,90.663,-177.8365,-0.3666,-15352.6841
C00568=55.455,-77.451,91.206,-179.0023,-0.8412,-15354.3973
C00569=53.310,-83.412,91.642,-179.7765,-0.5441,-15357.4167
C00570=48.140,-87.648,92.077,179.9985,-0.0384,-15361.2225
C00571=41.664,-90.907,92.362,179.9976,-0.0052,-15365.3773
C00572=34.820,-93.742,92.362,179.9980,-0.0054,-15369.6227
C00573=27.936,-96.017,92.077,-179.9986,-0.0362,-15373.7777
C00574=21.285,-96.677,91.642,179.7804,-0.5442,-15377.5835
C00575=15.553,-93.978,91.206,179.0014,-0.8397,-15380.6029
C00576=11.935,-88.455,90.663,177.8347,-0.3615,-15382.3156
C00577=10.790,-80.844,89.614,177.4669,-0.0031,-15382.3978
C00578=9.737,-72.291,87.405,177.2235,-0.0020,-15382.3289
C00579=8.774,-64.206,84.354,177.1343,-0.0134,-15382.2185
C00580=7.974,-57.808,81.229,177.8824,-0.0435,-15382.1462
C00581=6.711,-53.894,78.888,-169.2924,7.3770,-15382.9019
C00582=3.730,-52.747,77.945,-174.3297,24.7331,-15385.9551
C00583=1.476,-52.759,77.904,179.8644,26.2720,-15388.3975
C00584=0.000,-52.771,77.932,-180.0000,26.2576,-15390.0000
C00585=0.000,-52.771,77.932,-180.0000,26.2576,-15390.0000
C00586=-1.476,-52.759,77.904,-179.8644,26.2720,-15391.6025
C00587=-3.730,-52.747,77.945,174.3235,24.7327,-15394.0449
C00588=-6.711,-53.894,78.888,169.2924,7.3770,-15397.0981
C00589=-7.974,-57.808,81.229,-177.8824,-0.0435,-15397.8538
C00590=-8.774,-64.206,84.354,-177.1343,-0.0134,-15397.7815
C00591=-9.737,-72.291,87.405,-177.2235,-0.0020,-15397.6711
C00592=-10.790,-80.844,89.614,-177.4669,-0.0031,-15397.6022
C00593=-11.935,-88.455,90.663,-177.8347,-0.3615,-15397.6844
C00594=-15.553,-93.978,91.206,-179.0014,-0.8397,-15399.3971
C00595=-21.285,-96.677,91.642,-179.7804,-0.5442,-15402.4165
C00596=-27.936,-96.017,92.077,179.9986,-0.0362,-15406.2223
C00597=-34.820,-93.742,92.362,-179.9980,-0.0054,-15410.3773
C00598=-41.664,-90.907,92.362,-179.9976,-0.0052,-15414.6227
C00599=-48.140,-87.648,92.077,-179.9985,-0.0384,-15418.7775
C00600=-53.310,-83.412,91.642,179.7765,-0.5441,-15422.5833
C00601=-55.455,-77.451,91.206,179.0023,-0.8412,-15425.6027
C00602=-54.108,-70.986,90.663,177.8365,-0.3666,-15427.3159
C00603=-49.536,-64.795,89.614,177.4688,-0.0016,-15427.3980
C00604=-44.233,-58.003,87.405,177.2268,-0.0027,-15427.3291
C00605=-39.197,-51.604,84.354,177.1305,-0.0129,-15427.2193
C00606=-35.238,-46.514,81.229,177.8797,-0.0389,-15427.1468
C00607=-33.363,-42.854,78.888,-169.2963,7.3773,-15427.9017
C00608=-34.660,-39.935,77.945,-174.3268,24.7330,-15430.9551
C00609=-36.262,-38.350,77.904,179.8603,26.2704,-15433.3970
C00610=-37.314,-37.314,77.932,180.0000,26.2558,-15435.0000
C00611=-38.350,-36.262,77.904,-179.8603,26.2704,-15436.6030
C00612=-39.935,-34.660,77.945,174.3268,24.7330,-15439.0449
C00613=-42.854,-33.363,78.888,169.2928,7.3727,-15442.0983
C00614=-46.514,-35.238,81.229,-177.8797,-0.0389,-15442.8532
C00615=-51.604,-39.197,84.354,-177.1305,-0.0129,-15442.7807
C00616=-58.003,-44.233,87.405,-177.2268,-0.0027,-15442.6709
C00617=-64.795,-49.536,89.614,-177.4688,-0.0016,-15442.6020
C00618=-70.986,-54.108,90.663,-177.8365,-0.3666,-15442.6841
C00619=-77.451,-55.455,91.206,-179.0023,-0.8412,-15444.3973
C00620=-83.412,-53.310,91.642,-179.7765,-0.5441,-15447.4167
C00621=-87.648,-48.140,92.077,179.9985,-0.0384,-15451.2225
C00622=-90.907,-41.664,92.362,179.9976,-0.0052,-15455.3773
C00623=-93.742,-34.820,92.362,179.9980,-0.0054,-15459.6227
C00624=-96.017,-27.936,92.077,-179.9986,-0.0362,-15463.7777
C00625=-96.677,-21.285,91.642,179.7804,-0.5442,-15467.5835
C00626=-93.978,-15.553,91.206,179.0014,-0.8397,-15470.6029
C00627=-88.455,-11.935,90.663,177.8347,-0.3615,-15472.3156
C00628=-80.844,-10.790,89.614,177.4669,-0.0031,-15472.3978
C00629=-72.291,-9.737,87.405,177.2235,-0.0020,-15472.3289
C00630=-64.206,-8.774,84.354,177.1343,-0.0134,-15472.2185
C00631=-57.808,-7.974,81.229,177.8824,-0.0435,-15472.1462
C00632=-53.894,-6.711,78.888,-169.2924,7.3770,-15472.9019
C00633=-52.747,-3.730,77.945,-174.3297,24.7331,-15475.9551
C00634=-52.759,-1.476,77.904,179.8644,26.2720,-15478.3975
C00635=-52.771,0.000,77.932,-180.0000,26.2576,-15480.0000
C00636=-52.759,1.476,77.904,-179.8644,26.2720,-15481.6025
C00637=-52.747,3.730,77.945,174.3235,24.7327,-15484.0449
C00638=-53.894,6.711,78.888,169.2924,7.3770,-15487.0981
C00639=-57.808,7.974,81.229,-177.8824,-0.0435,-15487.8538
C00640=-64.206,8.774,84.354,-177.1343,-0.0134,-15487.7815
C00641=-72.291,9.737,87.405,-177.2235,-0.0020,-15487.6711
C00642=-80.844,10.790,89.614,-177.4669,-0.0031,-15487.6022
C00643=-88.455,11.935,90.663,-177.8347,-0.3615,-15487.6844
C00644=-93.978,15.553,91.206,-179.0014,-0.8397,-15489.3971
C00645=-96.677,21.285,91.642,-179.7804,-0.5442,-15492.4165
C00646=-96.017,27.936,92.077,179.9986,-0.0362,-15496.2223
C00647=-93.742,34.820,92.362,-179.9980,-0.0054,-15500.3773
C00648=-90.907,41.664,92.362,-179.9976,-0.0052,-15504.6227
C00649=-87.648,48.140,92.077,-179.9985,-0.0384,-15508.7775
C00650=-83.412,53.310,91.642,179.7765,-0.5441,-15512.5833
C00651=-77.451,55.455,91.206,179.0023,-0.8412,-15515.6027
C00652=-70.986,54.108,90.663,177.8365,-0.3666,-15517.3159
C00653=-64.795,49.536,89.614,177.4688,-0.0016,-15517.3980
C00654=-58.003,44.233,87.405,177.2268,-0.0027,-15517.3291
C00655=-51.604,39.197,84.354,177.1305,-0.0129,-15517.2193
C00656=-46.514,35.238,81.229,177.8797,-0.0389,-15517.1468
C00657=-42.854,33.363,78.888,-169.2963,7.3773,-15517.9017
C00658=-39.935,34.660,77.945,-174.3268,24.7330,-15520.9551
C00659=-38.350,36.262,77.904,179.8603,26.2704,-15523.3970
C00660=-37.314,37.314,77.932,180.0000,26.2558,-15525.0000
C00661=-36.262,38.350,77.904,-179.8603,26.2704,-15526.6030
C00662=-34.660,39.935,77.945,174.3268,24.7330,-15529.0449
C00663=-33.363,42.854,78.888,169.2928,7.3727,-15532.0983
C00664=-35.238,46.514,81.229,-177.8797,-0.0389,-15532.8532
C00665=-39.197,51.604,84.354,-177.1305,-0.0129,-15532.7807
C00666=-44.233,58.003,87.405,-177.2268,-0.0027,-15532.6709
C00667=-49.536,64.795,89.614,-177.4688,-0.0016,-15532.6020
C00668=-54.108,70.986,90.663,-177.8365,-0.3666,-15532.6841
C00669=-55.455,77.451,91.206,-179.0023,-0.8412,-15534.3973
C00670=-53.310,83.412,91.642,-179.7765,-0.5441,-15537.4167
C00671=-48.140,87.648,92.077,179.9985,-0.0384,-15541.2225
C00672=-41.664,90.907,92.362,179.9976,-0.0052,-15545.3773
C00673=-34.820,93.742,92.362,179.9980,-0.0054,-15549.6227
C00674=-27.936,96.017,92.077,-179.9986,-0.0362,-15553.7777
C00675=-21.285,96.677,91.642,179.7804,-0.5442,-15557.5835
C00676=-15.553,93.978,91.206,179.0014,-0.8397,-15560.6029
C00677=-11.935,88.455,90.663,177.8347,-0.3615,-15562.3156
C00678=-10.790,80.844,89.614,177.4669,-0.0031,-15562.3978
C00679=-9.737,72.291,87.405,177.2235,-0.0020,-15562.3289
C00680=-8.774,64.206,84.354,177.1343,-0.0134,-15562.2185
C00681=-7.974,57.808,81.229,177.8824,-0.0435,-15562.1462
C00682=-6.711,53.894,78.888,-169.2924,7.3770,-15562.9019
C00683=-3.730,52.747,77.945,-174.3235,24.7327,-15565.9551
C00684=-1.476,52.759,77.904,179.8644,26.2720,-15568.3975
C00685=0.000,52.771,77.932,-180.0000,26.2576,-15570.0000
C00686=0.000,51.832,79.921,-180.0000,24.1993,-15570.0000
C00687=1.391,51.822,79.893,-179.8934,24.2117,-15571.5376
C00688=3.586,51.820,79.935,174.6728,22.6760,-15573.9586
C00689=6.543,53.038,80.908,170.4732,6.3608,-15577.0327
C00690=7.793,57.125,83.313,-178.0121,-0.0296,-15577.7683
C00691=8.610,63.749,86.500,-177.5700,-0.0072,-15577.6919
C00692=9.608,72.041,89.587,-177.8667,0.0012,-15577.5966
C00693=10.692,80.728,91.809,-178.2949,0.0004,-15577.5446
C00694=11.850,88.408,92.861,-178.6931,-0.2180,-15577.6343
C00695=15.484,93.970,93.405,-179.4470,-0.4664,-15579.3569
C00696=21.237,96.685,93.841,-179.8869,-0.2743,-15582.3884
C00697=27.910,96.026,94.277,179.9993,-0.0181,-15586.2065
C00698=34.811,93.745,94.562,-180.0000,-0.0000,-15590.3718
C00699=41.672,90.903,94.562,-180.0000,-0.0000,-15594.6278
C00700=48.166,87.636,94.277,-179.9995,-0.0128,-15598.7938
C00701=53.350,83.383,93.841,179.8851,-0.2776,-15602.6119
C00702=55.498,77.395,93.405,179.4467,-0.4673,-15605.6434
C00703=54.135,70.893,92.861,178.6953,-0.2176,-15607.3659
C00704=49.523,64.644,91.809,178.2957,0.0009,-15607.4553
C00705=44.146,57.735,89.587,177.8657,-0.0015,-15607.4027
C00706=38.990,51.166,86.500,177.5699,-0.0071,-15607.3085
C00707=34.883,45.903,83.313,178.0127,-0.0275,-15607.2322
C00708=32.877,42.130,80.908,-170.4687,6.3616,-15607.9674
C00709=34.107,39.178,79.935,-174.6789,22.6775,-15611.0417
C00710=35.661,37.627,79.893,179.8957,24.2122,-15613.4634
C00711=36.651,36.651,79.921,180.0000,24.1961,-15615.0000
C00712=37.627,35.661,79.893,-179.8914,24.2160,-15616.5366
C00713=39.178,34.107,79.935,174.6702,22.6769,-15618.9583
C00714=42.130,32.877,80.908,170.4687,6.3616,-15622.0326
C00715=45.903,34.883,83.313,-178.0127,-0.0275,-15622.7678
C00716=51.166,38.990,86.500,-177.5699,-0.0071,-15622.6915
C00717=57.735,44.146,89.587,-177.8657,-0.0015,-15622.5973
C00718=64.644,49.523,91.809,-178.2957,0.0009,-15622.5447
C00719=70.893,54.135,92.861,-178.6953,-0.2176,-15622.6341
C00720=77.395,55.498,93.405,-179.4467,-0.4673,-15624.3566
C00721=83.383,53.350,93.841,-179.8851,-0.2776,-15627.3881
C00722=87.636,48.166,94.277,179.9995,-0.0128,-15631.2062
C00723=90.903,41.672,94.562,-180.0000,-0.0000,-15635.3722
C00724=93.745,34.811,94.562,-180.0000,-0.0000,-15639.6282
C00725=96.026,27.910,94.277,-179.9993,-0.0181,-15643.7935
C00726=96.685,21.237,93.841,179.8869,-0.2743,-15647.6116
C00727=93.970,15.484,93.405,179.4470,-0.4664,-15650.6431
C00728=88.408,11.850,92.861,178.6931,-0.2180,-15652.3657
C00729=80.728,10.692,91.809,178.2949,0.0004,-15652.4554
C00730=72.041,9.608,89.587,177.8667,0.0012,-15652.4034
C00731=63.749,8.610,86.500,177.5700,-0.0072,-15652.3081
C00732=57.125,7.793,83.313,178.0121,-0.0296,-15652.2317
C00733=53.038,6.543,80.908,-170.4732,6.3608,-15652.9673
C00734=51.820,3.586,79.935,-174.6728,22.6760,-15656.0414
C00735=51.822,1.391,79.893,179.8934,24.2117,-15658.4624
C00736=51.832,0.000,79.921,-180.0000,24.1993,-15660.0000
C00737=51.822,-1.390,79.893,-179.8929,24.2117,-15661.5365
C00738=51.820,-3.586,79.935,174.6728,22.6760,-15663.9586
C00739=53.038,-6.543,80.908,170.4732,6.3608,-15667.0327
C00740=57.125,-7.793,83.313,-178.0121,-0.0296,-15667.7683
C00741=63.749,-8.610,86.500,-177.5700,-0.0072,-15667.6919
C00742=72.041,-9.608,89.587,-177.8667,0.0012,-15667.5966
C00743=80.728,-10.692,91.809,-178.2949,0.0004,-15667.5446
C00744=88.408,-11.850,92.861,-178.6931,-0.2180,-15667.6343
C00745=93.970,-15.484,93.405,-179.4470,-0.4664,-15669.3569
C00746=96.685,-21.237,93.841,-179.8869,-0.2743,-15672.3884
C00747=96.026,-27.910,94.277,179.9993,-0.0181,-15676.2065
C00748=93.745,-34.811,94.562,-180.0000,-0.0000,-15680.3718
C00749=90.903,-41.672,94.562,-180.0000,-0.0000,-15684.6278
C00750=87.636,-48.166,94.277,-179.9995,-0.0128,-15688.7938
C00751=83.383,-53.350,93.841,179.8851,-0.2776,-15692.6119
C00752=77.395,-55.498,93.405,179.4467,-0.4673,-15695.6434
C00753=70.893,-54.135,92.861,178.6953,-0.2176,-15697.3659
C00754=64.644,-49.523,91.809,178.2957,0.0009,-15697.4553
C00755=57.735,-44.146,89.587,177.8657,-0.0015,-15697.4027
C00756=51.166,-38.990,86.500,177.5699,-0.0071,-15697.3085
C00757=45.903,-34.883,83.313,178.0127,-0.0275,-15697.2322
C00758=42.130,-32.877,80.908,-170.4687,6.3616,-15697.9674
C00759=39.178,-34.107,79.935,-174.6789,22.6775,-15701.0417
C00760=37.627,-35.661,79.893,179.8957,24.2122,-15703.4634
C00761=36.651,-36.651,79.921,-180.0000,24.1961,-15705.0000
C00762=35.661,-37.627,79.893,-179.8914,24.2160,-15706.5366
C00763=34.107,-39.178,79.935,174.6702,22.6769,-15708.9583
C00764=32.877,-42.130,80.908,170.4687,6.3616,-15712.0326
C00765=34.883,-45.903,83.313,-178.0127,-0.0275,-15712.7678
C00766=38.990,-51.166,86.500,-177.5699,-0.0071,-15712.6915
C00767=44.146,-57.735,89.587,-177.8657,-0.0015,-15712.5973
C00768=49.523,-64.644,91.809,-178.2957,0.0009,-15712.5447
C00769=54.135,-70.893,92.861,-178.6953,-0.2176,-15712.6341
C00770=55.498,-77.395,93.405,-179.4467,-0.4673,-15714.3566
C00771=53.350,-83.383,93.841,-179.8851,-0.2776,-15717.3881
C00772=48.166,-87.636,94.277,179.9995,-0.0128,-15721.2062
C00773=41.672,-90.903,94.562,-180.0000,-0.0000,-15725.3722
C00774=34.811,-93.745,94.562,-180.0000,-0.0000,-15729.6282
C00775=27.910,-96.026,94.277,-179.9993,-0.0181,-15733.7935
C00776=21.237,-96.685,93.841,179.8869,-0.2743,-15737.6116
C00777=15.484,-93.970,93.405,179.4470,-0.4664,-15740.6431
C00778=11.850,-88.408,92.861,178.6931,-0.2180,-15742.3657
C00779=10.692,-80.728,91.809,178.2949,0.0004,-15742.4554
C00780=9.608,-72.041,89.587,177.8667,0.0012,-15742.4034
C00781=8.610,-63.749,86.500,177.5700,-0.0072,-15742.3081
C00782=7.793,-57.125,83.313,178.0121,-0.0296,-15742.2317
C00783=6.543,-53.038,80.908,-170.4732,6.3608,-15742.9673
C00784=3.586,-51.820,79.935,-174.6728,22.6760,-15746.0414
C00785=1.391,-51.822,79.893,179.8934,24.2117,-15748.4624
C00786=0.000,-51.832,79.921,180.0000,24.1993,-15750.0000
C00787=0.000,-51.832,79.921,180.0000,24.1993,-15750.0000
C00788=-1.390,-51.822,79.893,-179.8929,24.2117,-15751.5365
C00789=-3.586,-51.820,79.935,174.6728,22.6760,-15753.9586
C00790=-6.543,-53.038,80.908,170.4732,6.3608,-15757.0327
C00791=-7.793,-57.125,83.313,-178.0121,-0.0296,-15757.7683
C00792=-8.610,-63.749,86.500,-177.5700,-0.0072,-15757.6919
C00793=-9.608,-72.041,89.587,-177.8667,0.0012,-15757.5966
C00794=-10.692,-80.728,91.809,-178.2949,0.0004,-15757.5446
C00795=-11.850,-88.408,92.861,-178.6931,-0.2180,-15757.6343
C00796=-15.484,-93.970,93.405,-179.4470,-0.4664,-15759.3569
C00797=-21.237,-96.685,93.841,-179.8869,-0.2743,-15762.3884
C00798=-27.910,-96.026,94.277,179.9993,-0.0181,-15766.2065
C00799=-34.811,-93.745,94.562,-180.0000,-0.0000,-15770.3718
C00800=-41.672,-90.903,94.562,-180.0000,-0.0000,-15774.6278
C00801=-48.166,-87.636,94.277,-179.9995,-0.0128,-15778.7938
C00802=-53.350,-83.383,93.841,179.8851,-0.2776,-15782.6119
C00803=-55.498,-77.395,93.405,179.4467,-0.4673,-15785.6434
C00804=-54.135,-70.893,92.861,178.6953,-0.2176,-15787.3659
C00805=-49.523,-64.644,91.809,178.2957,0.0009,-15787.4553
C00806=-44.146,-57.735,89.587,177.8657,-0.0015,-15787.4027
C00807=-38.990,-51.166,86.500,177.5699,-0.0071,-15787.3085
C00808=-34.883,-45.903,83.313,178.0127,-0.0275,-15787.2322
C00809=-32.877,-42.130,80.908,-170.4687,6.3616,-15787.9674
C00810=-34.107,-39.178,79.935,-174.6789,22.6775,-15791.0417
C00811=-35.661,-37.627,79.893,179.8957,24.2122,-15793.4634
C00812=-36.651,-36.651,79.921,-180.0000,24.1961,-15795.0000
C00813=-37.627,-35.661,79.893,-179.8914,24.2160,-15796.5366
C00814=-39.178,-34.107,79.935,174.6702,22.6769,-15798.9583
C00815=-42.130,-32.877,80.908,170.4687,6.3616,-15802.0326
C00816=-45.903,-34.883,83.313,-178.0127,-0.0275,-15802.7678
C00817=-51.166,-38.990,86.500,-177.5699,-0.0071,-15802.6915
C00818=-57.735,-44.146,89.587,-177.8657,-0.0015,-15802.5973
C00819=-64.644,-49.523,91.809,-178.2957,0.0009,-15802.5447
C00820=-70.893,-54.135,92.861,-178.6953,-0.2176,-15802.6341
C00821=-77.395,-55.498,93.405,-179.4467,-0.4673,-15804.3566
C00822=-83.383,-53.350,93.841,-179.8851,-0.2776,-15807.3881
C00823=-87.636,-48.166,94.277,179.9995,-0.0128,-15811.2062
C00824=-90.903,-41.672,94.562,-180.0000,-0.0000,-15815.3722
C00825=-93.745,-34.811,94.562,-180.0000,-0.0000,-15819.6282
C00826=-96.026,-27.910,94.277,-179.9993,-0.0181,-15823.7935
C00827=-96.685,-21.237,93.841,179.8869,-0.2743,-15827.6116
C00828=-93.970,-15.484,93.405,179.4470,-0.4664,-15830.6431
C00829=-88.408,-11.850,92.861,178.6931,-0.2180,-15832.3657
C00830=-80.728,-10.692,91.809,178.2949,0.0004,-15832.4554
C00831=-72.041,-9.608,89.587,177.8667,0.0012,-15832.4034
C00832=-63.749,-8.610,86.500,177.5700,-0.0072,-15832.3081
C00833=-57.125,-7.793,83.313,178.0121,-0.0296,-15832.2317
C00834=-53.038,-6.543,80.908,-170.4732,6.3608,-15832.9673
C00835=-51.820,-3.586,79.935,-174.6728,22.6760,-15836.0414
C00836=-51.822,-1.391,79.893,179.8934,24.2117,-15838.4624
C00837=-51.832,0.000,79.921,180.0000,24.1993,-15840.0000
C00838=-51.822,1.390,79.893,-179.8929,24.2117,-15841.5365
C00839=-51.820,3.586,79.935,174.6728,22.6760,-15843.9586
C00840=-53.038,6.543,80.908,170.4732,6.3608,-15847.0327
C00841=-57.125,7.793,83.313,-178.0121,-0.0296,-15847.7683
C00842=-63.749,8.610,86.500,-177.5700,-0.0072,-15847.6919
C00843=-72.041,9.608,89.587,-177.8667,0.0012,-15847.5966
C00844=-80.728,10.692,91.809,-178.2949,0.0004,-15847.5446
C00845=-88.408,11.850,92.861,-178.6931,-0.2180,-15847.6343
C00846=-93.970,15.484,93.405,-179.4470,-0.4664,-15849.3569
C00847=-96.685,21.237,93.841,-179.8869,-0.2743,-15852.3884
C00848=-96.026,27.910,94.277,179.9993,-0.0181,-15856.2065
C00849=-93.745,34.811,94.562,-180.0000,-0.0000,-15860.3718
C00850=-90.903,41.672,94.562,-180.0000,-0.0000,-15864.6278
C00851=-87.636,48.166,94.277,-179.9995,-0.0128,-15868.7938
C00852=-83.383,53.350,93.841,179.8851,-0.2776,-15872.6119
C00853=-77.395,55.498,93.405,179.4467,-0.4673,-15875.6434
C00854=-70.893,54.135,92.861,178.6953,-0.2176,-15877.3659
C00855=-64.644,49.523,91.809,178.2957,0.0009,-15877.4553
C00856=-57.735,44.146,89.587,177.8657,-0.0015,-15877.4027
C00857=-51.166,38.990,86.500,177.5699,-0.0071,-15877.3085
C00858=-45.903,34.883,83.313,178.0127,-0.0275,-15877.2322
C00859=-42.130,32.877,80.908,-170.4687,6.3616,-15877.9674
C00860=-39.178,34.107,79.935,-174.6789,22.6775,-15881.0417
C00861=-37.627,35.661,79.893,179.8957,24.2122,-15883.4634
C00862=-36.651,36.651,79.921,-180.0000,24.1961,-15885.0000
C00863=-35.661,37.627,79.893,-179.8914,24.2160,-15886.5366
C00864=-34.107,39.178,79.935,174.6702,22.6769,-15888.9583
C00865=-32.877,42.130,80.908,170.4687,6.3616,-15892.0326
C00866=-34.883,45.903,83.313,-178.0127,-0.0275,-15892.7678
C00867=-38.990,51.166,86.500,-177.5699,-0.0071,-15892.6915
C00868=-44.146,57.735,89.587,-177.8657,-0.0015,-15892.5973
C00869=-49.523,64.644,91.809,-178.2957,0.0009,-15892.5447
C00870=-54.135,70.893,92.861,-178.6953,-0.2176,-15892.6341
C00871=-55.498,77.395,93.405,-179.4467,-0.4673,-15894.3566
C00872=-53.350,83.383,93.841,-179.8851,-0.2776,-15897.3881
C00873=-48.166,87.636,94.277,179.9995,-0.0128,-15901.2062
C00874=-41.672,90.903,94.562,-180.0000,-0.0000,-15905.3722
C00875=-34.811,93.745,94.562,-180.0000,-0.0000,-15909.6282
C00876=-27.910,96.026,94.277,-179.9993,-0.0181,-15913.7935
C00877=-21.237,96.685,93.841,179.8869,-0.2743,-15917.6116
C00878=-15.484,93.970,93.405,179.4470,-0.4664,-15920.6431
C00879=-11.850,88.408,92.861,178.6931,-0.2180,-15922.3657
C00880=-10.692,80.728,91.809,178.2949,0.0004,-15922.4554
C00881=-9.608,72.041,89.587,177.8667,0.0012,-15922.4034
C00882=-8.610,63.749,86.500,177.5700,-0.0072,-15922.3081
C00883=-7.793,57.125,83.313,178.0121,-0.0296,-15922.2317
C00884=-6.543,53.038,80.908,-170.4732,6.3608,-15922.9673
C00885=-3.586,51.820,79.935,-174.6728,22.6760,-15926.0414
C00886=-1.390,51.822,79.893,179.8929,24.2117,-15928.4635
C00887=0.000,51.832,79.921,180.0000,24.1993,-15930.0000
C00888=0.000,50.970,81.946,180.0000,21.8993,-15930.0000
C00889=1.312,50.962,81.916,-179.9262,21.9171,-15931.4747
C00890=3.453,50.970,81.960,175.1064,20.4142,-15933.8756
C00891=6.389,52.261,82.960,171.6928,5.3944,-15936.9699
C00892=7.633,56.525,85.423,-178.2163,-0.0194,-15937.6906
C00893=8.475,63.374,88.663,-178.0565,-0.0061,-15937.6170
C00894=9.515,71.858,91.777,-178.5551,0.0006,-15937.5429
C00895=10.634,80.658,94.007,-179.1678,-0.0001,-15937.5106
C00896=11.808,88.386,95.061,-179.5979,-0.0677,-15937.6094
C00897=15.455,93.966,95.604,-179.9126,-0.0727,-15939.3401
C00898=55.516,77.372,95.604,179.9102,-0.0715,-15965.6602
C00899=54.149,70.847,95.061,179.5984,-0.0690,-15967.3910
C00900=49.515,64.553,94.007,179.1703,-0.0010,-15967.4898
C00901=44.083,57.539,91.777,178.5571,-0.0010,-15967.4572
C00902=38.820,50.805,88.663,178.0538,-0.0014,-15967.3834
C00903=34.571,45.367,85.423,178.2190,-0.0171,-15967.3085
C00904=32.436,41.472,82.960,-171.6874,5.3944,-15968.0296
C00905=33.599,38.483,81.960,-175.1072,20.4131,-15971.1238
C00906=35.108,36.963,81.916,179.9250,21.9192,-15973.5256
C00907=36.041,36.041,81.946,-180.0000,21.8955,-15975.0000
C00908=36.963,35.108,81.916,-179.9250,21.9192,-15976.4744
C00909=38.483,33.599,81.960,175.1072,20.4131,-15978.8762
C00910=41.472,32.436,82.960,171.6919,5.3909,-15981.9704
C00911=45.367,34.571,85.423,-178.2190,-0.0171,-15982.6915
C00912=50.805,38.820,88.663,-178.0538,-0.0014,-15982.6166
C00913=57.539,44.083,91.777,-178.5571,-0.0010,-15982.5428
C00914=64.553,49.515,94.007,-179.1703,-0.0010,-15982.5102
C00915=70.847,54.149,95.061,-179.5984,-0.0690,-15982.6090
C00916=77.372,55.516,95.604,-179.9102,-0.0715,-15984.3398
C00917=93.966,15.455,95.604,179.9126,-0.0727,-16010.6599
C00918=88.386,11.808,95.061,179.5979,-0.0677,-16012.3906
C00919=80.658,10.634,94.007,179.1678,-0.0001,-16012.4894
C00920=71.858,9.515,91.777,178.5551,0.0006,-16012.4571
C00921=63.374,8.475,88.663,178.0565,-0.0061,-16012.3830
C00922=56.525,7.633,85.423,178.2163,-0.0194,-16012.3094
C00923=52.261,6.389,82.960,-171.6928,5.3944,-16013.0301
C00924=50.970,3.453,81.960,-175.1064,20.4142,-16016.1244
C00925=50.962,1.312,81.916,179.9262,21.9171,-16018.5253
C00926=50.970,0.000,81.946,180.0000,21.8993,-16020.0000
C00927=50.962,-1.311,81.916,-179.9258,21.9171,-16021.4736
C00928=50.970,-3.454,81.960,175.1060,20.4141,-16023.8767
C00929=52.261,-6.389,82.960,171.6928,5.3944,-16026.9699
C00930=56.525,-7.633,85.423,-178.2163,-0.0194,-16027.6906
C00931=63.374,-8.475,88.663,-178.0565,-0.0061,-16027.6170
C00932=71.858,-9.515,91.777,-178.5551,0.0006,-16027.5429
C00933=80.658,-10.634,94.007,-179.1678,-0.0001,-16027.5106
C00934=88.386,-11.808,95.061,-179.5979,-0.0677,-16027.6094
C00935=93.966,-15.455,95.604,-179.9126,-0.0727,-16029.3401
C00936=77.372,-55.516,95.604,179.9102,-0.0715,-16055.6602
C00937=70.847,-54.149,95.061,179.5984,-0.0690,-16057.3910
C00938=64.553,-49.515,94.007,179.1703,-0.0010,-16057.4898
C00939=57.539,-44.083,91.777,178.5571,-0.0010,-16057.4572
C00940=50.805,-38.820,88.663,178.0538,-0.0014,-16057.3834
C00941=45.367,-34.571,85.423,178.2190,-0.0171,-16057.3085
C00942=41.472,-32.436,82.960,-171.6874,5.3944,-16058.0296
C00943=38.483,-33.599,81.960,-175.1072,20.4131,-16061.1238
C00944=36.963,-35.108,81.916,179.9250,21.9192,-16063.5256
C00945=36.041,-36.041,81.946,-180.0000,21.8955,-16065.0000
C00946=35.108,-36.963,81.916,-179.9250,21.9192,-16066.4744
C00947=33.599,-38.483,81.960,175.1072,20.4131,-16068.8762
C00948=32.436,-41.472,82.960,171.6919,5.3909,-16071.9704
C00949=34.571,-45.367,85.423,-178.2190,-0.0171,-16072.6915
C00950=38.820,-50.805,88.663,-178.0538,-0.0014,-16072.6166
C00951=44.083,-57.539,91.777,-178.5571,-0.0010,-16072.5428
C00952=49.515,-64.553,94.007,-179.1703,-0.0010,-16072.5102
C00953=54.149,-70.847,95.061,-179.5984,-0.0690,-16072.6090
C00954=55.516,-77.372,95.604,-179.9102,-0.0715,-16074.3398
C00955=15.455,-93.966,95.604,179.9126,-0.0727,-16100.6599
C00956=11.808,-88.386,95.061,179.5979,-0.0677,-16102.3906
C00957=10.634,-80.658,94.007,179.1678,-0.0001,-16102.4894
C00958=9.515,-71.858,91.777,178.5551,0.0006,-16102.4571
C00959=8.475,-63.374,88.663,178.0565,-0.0061,-16102.3830
C00960=7.633,-56.525,85.423,178.2163,-0.0194,-16102.3094
C00961=6.389,-52.261,82.960,-171.6928,5.3944,-16103.0301
C00962=3.453,-50.970,81.960,-175.1064,20.4142,-16106.1244
C00963=1.312,-50.962,81.916,179.9262,21.9171,-16108.5253
C00964=0.000,-50.970,81.946,180.0000,21.8993,-16110.0000
C00965=0.000,-50.970,81.946,180.0000,21.8993,-16110.0000
C00966=-1.311,-50.962,81.916,-179.9258,21.9171,-16111.4736
C00967=-3.454,-50.970,81.960,175.1060,20.4141,-16113.8767
C00968=-6.389,-52.261,82.960,171.6928,5.3944,-16116.9699
C00969=-7.633,-56.525,85.423,-178.2163,-0.0194,-16117.6906
C00970=-8.475,-63.374,88.663,-178.0565,-0.0061,-16117.6170
C00971=-9.515,-71.858,91.777,-178.5551,0.0006,-16117.5429
C00972=-10.634,-80.658,94.007,-179.1678,-0.0001,-16117.5106
C00973=-11.808,-88.386,95.061,-179.5979,-0.0677,-16117.6094
C00974=-15.455,-93.966,95.604,-179.9126,-0.0727,-16119.3401
C00975=-55.516,-77.372,95.604,179.9102,-0.0715,-16145.6602
C00976=-54.149,-70.847,95.061,179.5984,-0.0690,-16147.3910
C00977=-49.515,-64.553,94.007,179.1703,-0.0010,-16147.4898
C00978=-44.083,-57.539,91.777,178.5571,-0.0010,-16147.4572
C00979=-38.820,-50.805,88.663,178.0538,-0.0014,-16147.3834
C00980=-34.571,-45.367,85.423,178.2190,-0.0171,-16147.3085
C00981=-32.436,-41.472,82.960,-171.6874,5.3944,-16148.0296
C00982=-33.599,-38.483,81.960,-175.1072,20.4131,-16151.1238
C00983=-35.108,-36.963,81.916,179.9250,21.9192,-16153.5256
C00984=-36.041,-36.041,81.946,-180.0000,21.8955,-16155.0000
C00985=-36.963,-35.108,81.916,-179.9250,21.9192,-16156.4744
C00986=-38.483,-33.599,81.960,175.1072,20.4131,-16158.8762
C00987=-41.472,-32.436,82.960,171.6919,5.3909,-16161.9704
C00988=-45.367,-34.571,85.423,-178.2190,-0.0171,-16162.6915
C00989=-50.805,-38.820,88.663,-178.0538,-0.0014,-16162.6166
C00990=-57.539,-44.083,91.777,-178.5571,-0.0010,-16162.5428
C00991=-64.553,-49.515,94.007,-179.1703,-0.0010,-16162.5102
C00992=-70.847,-54.149,95.061,-179.5984,-0.0690,-16162.6090
C00993=-77.372,-55.516,95.604,-179.9102,-0.0715,-16164.3398
C00994=-93.966,-15.455,95.604,179.9126,-0.0727,-16190.6599
C00995=-88.386,-11.808,95.061,179.5979,-0.0677,-16192.3906
C00996=-80.658,-10.634,94.007,179.1678,-0.0001,-16192.4894
C00997=-71.858,-9.515,91.777,178.5551,0.0006,-16192.4571
C00998=-63.374,-8.475,88.663,178.0565,-0.0061,-16192.3830
C00999=-56.525,-7.633,85.423,178.2163,-0.0194,-16192.3094
C01000=-52.261,-6.389,82.960,-171.6928,5.3944,-16193.0301
C01001=-50.970,-3.453,81.960,-175.1064,20.4142,-16196.1244
C01002=-50.962,-1.312,81.916,179.9262,21.9171,-16198.5253
C01003=-50.970,0.000,81.946,-180.0000,21.8993,-16200.0000
C01004=-50.962,1.311,81.916,-179.9258,21.9171,-16201.4736
C01005=-50.970,3.454,81.960,175.1060,20.4141,-16203.8767
C01006=-52.261,6.389,82.960,171.6928,5.3944,-16206.9699
C01007=-56.525,7.633,85.423,-178.2163,-0.0194,-16207.6906
C01008=-63.374,8.475,88.663,-178.0565,-0.0061,-16207.6170
C01009=-71.858,9.515,91.777,-178.5551,0.0006,-16207.5429
C01010=-80.658,10.634,94.007,-179.1678,-0.0001,-16207.5106
C01011=-88.386,11.808,95.061,-179.5979,-0.0677,-16207.6094
C01012=-93.966,15.455,95.604,-179.9126,-0.0727,-16209.3401
C01013=-77.372,55.516,95.604,179.9102,-0.0715,-16235.6602
C01014=-70.847,54.149,95.061,179.5984,-0.0690,-16237.3910
C01015=-64.553,49.515,94.007,179.1703,-0.0010,-16237.4898
C01016=-57.539,44.083,91.777,178.5571,-0.0010,-16237.4572
C01017=-50.805,38.820,88.663,178.0538,-0.0014,-16237.3834
C01018=-45.367,34.571,85.423,178.2190,-0.0171,-16237.3085
C01019=-41.472,32.436,82.960,-171.6874,5.3944,-16238.0296
C01020=-38.483,33.599,81.960,-175.1072,20.4131,-16241.1238
C01021=-36.963,35.108,81.916,179.9250,21.9192,-16243.5256
C01022=-36.041,36.041,81.946,180.0000,21.8955,-16245.0000
C01023=-35.108,36.963,81.916,-179.9250,21.9192,-16246.4744
C01024=-33.599,38.483,81.960,175.1072,20.4131,-16248.8762
C01025=-32.436,41.472,82.960,171.6919,5.3909,-16251.9704
C01026=-34.571,45.367,85.423,-178.2190,-0.0171,-16252.6915
C01027=-38.820,50.805,88.663,-178.0538,-0.0014,-16252.6166
C01028=-44.083,57.539,91.777,-178.5571,-0.0010,-16252.5428
C01029=-49.515,64.553,94.007,-179.1703,-0.0010,-16252.5102
C01030=-54.149,70.847,95.061,-179.5984,-0.0690,-16252.6090
C01031=-55.516,77.372,95.604,-179.9102,-0.0715,-16254.3398
C01032=-15.455,93.966,95.604,179.9126,-0.0727,-16280.6599
C01033=-11.808,88.386,95.061,179.5979,-0.0677,-16282.3906
C01034=-10.634,80.658,94.007,179.1678,-0.0001,-16282.4894
C01035=-9.515,71.858,91.777,178.5551,0.0006,-16282.4571
C01036=-8.475,63.374,88.663,178.0565,-0.0061,-16282.3830
C01037=-7.633,56.525,85.423,178.2163,-0.0194,-16282.3094
C01038=-6.389,52.261,82.960,-171.6928,5.3944,-16283.0301
C01039=-3.454,50.970,81.960,-175.1060,20.4141,-16286.1233
C01040=-1.311,50.962,81.916,179.9258,21.9171,-16288.5264
C01041=0.000,50.970,81.946,-180.0000,21.8993,-16290.0000
C01042=0.000,50.195,84.004,-180.0000,19.3355,-16290.0000
C01043=1.241,50.188,83.974,-179.9511,19.3601,-16291.4165
C01044=3.334,50.204,84.019,175.6244,17.9316,-16293.7994
C01045=6.253,51.571,85.045,172.9492,4.4629,-16296.9134
C01046=7.499,56.017,87.559,-178.4839,-0.0109,-16297.6249
C01047=8.371,63.087,90.842,-178.5891,-0.0035,-16297.5584
C01048=9.459,71.748,93.974,-179.2893,0.0012,-16297.5104
C01049=44.045,57.421,93.974,179.2929,-0.0008,-16327.4901
C01050=38.690,50.529,90.842,178.5857,-0.0004,-16327.4412
C01051=34.307,44.912,87.559,178.4862,-0.0099,-16327.3752
C01052=32.045,40.888,85.045,-172.9480,4.4644,-16328.0867
C01053=33.142,37.857,84.019,-175.6236,17.9314,-16331.2006
C01054=34.611,36.365,83.974,179.9520,19.3612,-16333.5844
C01055=35.493,35.493,84.004,179.9957,19.3375,-16335.0000
C01056=36.365,34.611,83.974,-179.9520,19.3612,-16336.4156
C01057=37.858,33.142,84.019,175.6234,17.9313,-16338.8001
C01058=40.888,32.045,85.045,172.9480,4.4644,-16341.9133
C01059=44.912,34.307,87.559,-178.4862,-0.0099,-16342.6248
C01060=50.529,38.690,90.842,-178.5857,-0.0004,-16342.5588
C01061=57.421,44.045,93.974,-179.2929,-0.0008,-16342.5099
C01062=71.748,9.459,93.974,179.2893,0.0012,-16372.4896
C01063=63.087,8.371,90.842,178.5891,-0.0035,-16372.4416
C01064=56.017,7.499,87.559,178.4839,-0.0109,-16372.3751
C01065=51.571,6.253,85.045,-172.9492,4.4629,-16373.0866
C01066=50.204,3.334,84.019,-175.6244,17.9316,-16376.2006
C01067=50.188,1.241,83.974,179.9511,19.3601,-16378.5835
C01068=50.195,0.000,84.004,-180.0000,19.3355,-16380.0000
C01069=50.188,-1.240,83.974,-179.9507,19.3601,-16381.4153
C01070=50.204,-3.335,84.019,175.6241,17.9315,-16383.8005
C01071=51.571,-6.253,85.045,172.9492,4.4629,-16386.9134
C01072=56.017,-7.499,87.559,-178.4839,-0.0109,-16387.6249
C01073=63.087,-8.371,90.842,-178.5891,-0.0035,-16387.5584
C01074=71.748,-9.459,93.974,-179.2893,0.0012,-16387.5104
C01075=57.421,-44.045,93.974,179.2929,-0.0008,-16417.4901
C01076=50.529,-38.690,90.842,178.5857,-0.0004,-16417.4412
C01077=44.912,-34.307,87.559,178.4862,-0.0099,-16417.3752
C01078=40.888,-32.045,85.045,-172.9480,4.4644,-16418.0867
C01079=37.857,-33.142,84.019,-175.6236,17.9314,-16421.2006
C01080=36.365,-34.611,83.974,179.9520,19.3612,-16423.5844
C01081=35.493,-35.493,84.004,179.9957,19.3375,-16425.0000
C01082=34.611,-36.365,83.974,-179.9520,19.3612,-16426.4156
C01083=33.142,-37.858,84.019,175.6234,17.9313,-16428.8001
C01084=32.045,-40.888,85.045,172.9480,4.4644,-16431.9133
C01085=34.307,-44.912,87.559,-178.4862,-0.0099,-16432.6248
C01086=38.690,-50.529,90.842,-178.5857,-0.0004,-16432.5588
C01087=44.045,-57.421,93.974,-179.2929,-0.0008,-16432.5099
C01088=9.459,-71.748,93.974,179.2893,0.0012,-16462.4896
C01089=8.371,-63.087,90.842,178.5891,-0.0035,-16462.4416
C01090=7.499,-56.017,87.559,178.4839,-0.0109,-16462.3751
C01091=6.253,-51.571,85.045,-172.9492,4.4629,-16463.0866
C01092=3.334,-50.204,84.019,-175.6244,17.9316,-16466.2006
C01093=1.241,-50.188,83.974,179.9511,19.3601,-16468.5835
C01094=0.000,-50.195,84.004,-180.0000,19.3355,-16470.0000
C01095=0.000,-50.195,84.004,-180.0000,19.3355,-16470.0000
C01096=-1.240,-50.188,83.974,-179.9507,19.3601,-16471.4153
C01097=-3.335,-50.204,84.019,175.6241,17.9315,-16473.8005
C01098=-6.253,-51.571,85.045,172.9492,4.4629,-16476.9134
C01099=-7.499,-56.017,87.559,-178.4839,-0.0109,-16477.6249
C01100=-8.371,-63.087,90.842,-178.5891,-0.0035,-16477.5584
C01101=-9.459,-71.748,93.974,-179.2893,0.0012,-16477.5104
C01102=-44.045,-57.421,93.974,179.2929,-0.0008,-16507.4901
C01103=-38.690,-50.529,90.842,178.5857,-0.0004,-16507.4412
C01104=-34.307,-44.912,87.559,178.4862,-0.0099,-16507.3752
C01105=-32.045,-40.888,85.045,-172.9480,4.4644,-16508.0867
C01106=-33.142,-37.857,84.019,-175.6236,17.9314,-16511.2006
C01107=-34.611,-36.365,83.974,179.9520,19.3612,-16513.5844
C01108=-35.493,-35.493,84.004,179.9957,19.3375,-16515.0000
C01109=-36.365,-34.611,83.974,-179.9520,19.3612,-16516.4156
C01110=-37.858,-33.142,84.019,175.6234,17.9313,-16518.8001
C01111=-40.888,-32.045,85.045,172.9480,4.4644,-16521.9133
C01112=-44.912,-34.307,87.559,-178.4862,-0.0099,-16522.6248
C01113=-50.529,-38.690,90.842,-178.5857,-0.0004,-16522.5588
C01114=-57.421,-44.045,93.974,-179.2929,-0.0008,-16522.5099
C01115=-71.748,-9.459,93.974,179.2893,0.0012,-16552.4896
C01116=-63.087,-8.371,90.842,178.5891,-0.0035,-16552.4416
C01117=-56.017,-7.499,87.559,178.4839,-0.0109,-16552.3751
C01118=-51.571,-6.253,85.045,-172.9492,4.4629,-16553.0866
C01119=-50.204,-3.334,84.019,-175.6244,17.9316,-16556.2006
C01120=-50.188,-1.241,83.974,179.9511,19.3601,-16558.5835
C01121=-50.195,0.000,84.004,-180.0000,19.3355,-16560.0000
C01122=-50.188,1.240,83.974,-179.9507,19.3601,-16561.4153
C01123=-50.204,3.335,84.019,175.6241,17.9315,-16563.8005
C01124=-51.571,6.253,85.045,172.9492,4.4629,-16566.9134
C01125=-56.017,7.499,87.559,-178.4839,-0.0109,-16567.6249
C01126=-63.087,8.371,90.842,-178.5891,-0.0035,-16567.5584
C01127=-71.748,9.459,93.974,-179.2893,0.0012,-16567.5104
C01128=-57.421,44.045,93.974,179.2929,-0.0008,-16597.4901
C01129=-50.529,38.690,90.842,178.5857,-0.0004,-16597.4412
C01130=-44.912,34.307,87.559,178.4862,-0.0099,-16597.3752
C01131=-40.888,32.045,85.045,-172.9480,4.4644,-16598.0867
C01132=-37.857,33.142,84.019,-175.6236,17.9314,-16601.2006
C01133=-36.365,34.611,83.974,179.9520,19.3612,-16603.5844
C01134=-35.493,35.493,84.004,179.9957,19.3375,-16605.0000
C01135=-34.611,36.365,83.974,-179.9520,19.3612,-16606.4156
C01136=-33.142,37.858,84.019,175.6234,17.9313,-16608.8001
C01137=-32.045,40.888,85.045,172.9480,4.4644,-16611.9133
C01138=-34.307,44.912,87.559,-178.4862,-0.0099,-16612.6248
C01139=-38.690,50.529,90.842,-178.5857,-0.0004,-16612.5588
C01140=-44.045,57.421,93.974,-179.2929,-0.0008,-16612.5099
C01141=-9.459,71.748,93.974,179.2893,0.0012,-16642.4896
C01142=-8.371,63.087,90.842,178.5891,-0.0035,-16642.4416
C01143=-7.499,56.017,87.559,178.4839,-0.0109,-16642.3751
C01144=-6.253,51.571,85.045,-172.9492,4.4629,-16643.0866
C01145=-3.335,50.204,84.019,-175.6241,17.9315,-16646.1995
C01146=-1.240,50.188,83.974,179.9507,19.3601,-16648.5847
C01147=0.000,50.195,84.004,-180.0000,19.3355,-16650.0000
C01148=0.000,49.517,86.097,-180.0000,16.4995,-16650.0000
C01149=1.179,49.510,86.067,-179.9745,16.5281,-16651.3641
C01150=3.230,49.536,86.112,176.2280,15.2268,-16653.7307
C01151=6.137,50.981,87.161,174.2492,3.5661,-16656.8641
C01152=7.391,55.610,89.719,-178.8088,-0.0035,-16657.5707
C01153=8.302,62.896,93.033,-179.1621,0.0008,-16657.5193
C01154=38.603,50.345,93.033,179.1623,0.0002,-16687.4799
C01155=34.096,44.548,89.719,178.8104,-0.0013,-16687.4296
C01156=31.710,40.389,87.161,-174.2479,3.5658,-16688.1360
C01157=32.743,37.311,86.112,-176.2272,15.2245,-16691.2692
C01158=34.176,35.843,86.067,179.9736,16.5280,-16693.6362
C01159=35.014,35.014,86.097,179.9958,16.5019,-16695.0000
C01160=35.842,34.176,86.067,-179.9734,16.5280,-16696.3630
C01161=37.311,32.743,86.112,176.2272,15.2245,-16698.7308
C01162=40.389,31.710,87.161,174.2524,3.5623,-16701.8640
C01163=44.548,34.096,89.719,-178.8104,-0.0013,-16702.5704
C01164=50.345,38.603,93.033,-179.1623,0.0002,-16702.5201
C01165=62.896,8.302,93.033,179.1621,0.0008,-16732.4807
C01166=55.610,7.391,89.719,178.8088,-0.0035,-16732.4293
C01167=50.981,6.137,87.161,-174.2492,3.5661,-16733.1359
C01168=49.536,3.230,86.112,-176.2280,15.2268,-16736.2693
C01169=49.510,1.179,86.067,179.9745,16.5281,-16738.6359
C01170=49.517,0.000,86.097,180.0000,16.4995,-16740.0000
C01171=49.510,-1.178,86.067,-179.9741,16.5281,-16741.3630
C01172=49.536,-3.231,86.112,176.2280,15.2212,-16743.7318
C01173=50.981,-6.137,87.161,174.2492,3.5661,-16746.8641
C01174=55.610,-7.391,89.719,-178.8088,-0.0035,-16747.5707
C01175=62.896,-8.302,93.033,-179.1621,0.0008,-16747.5193
C01176=50.345,-38.603,93.033,179.1623,0.0002,-16777.4799
C01177=44.548,-34.096,89.719,178.8104,-0.0013,-16777.4296
C01178=40.389,-31.710,87.161,-174.2479,3.5658,-16778.1360
C01179=37.311,-32.743,86.112,-176.2272,15.2245,-16781.2692
C01180=35.843,-34.176,86.067,179.9736,16.5280,-16783.6362
C01181=35.014,-35.014,86.097,179.9958,16.5019,-16785.0000
C01182=34.176,-35.842,86.067,-179.9734,16.5280,-16786.3630
C01183=32.743,-37.311,86.112,176.2272,15.2245,-16788.7308
C01184=31.710,-40.389,87.161,174.2524,3.5623,-16791.8640
C01185=34.096,-44.548,89.719,-178.8104,-0.0013,-16792.5704
C01186=38.603,-50.345,93.033,-179.1623,0.0002,-16792.5201
C01187=8.302,-62.896,93.033,179.1621,0.0008,-16822.4807
C01188=7.391,-55.610,89.719,178.8088,-0.0035,-16822.4293
C01189=6.137,-50.981,87.161,-174.2492,3.5661,-16823.1359
C01190=3.230,-49.536,86.112,-176.2280,15.2268,-16826.2693
C01191=1.179,-49.510,86.067,179.9745,16.5281,-16828.6359
C01192=0.000,-49.517,86.097,180.0000,16.4995,-16830.0000
C01193=0.000,-49.517,86.097,180.0000,16.4995,-16830.0000
C01194=-1.178,-49.510,86.067,-179.9741,16.5281,-16831.3630
C01195=-3.231,-49.536,86.112,176.2280,15.2212,-16833.7318
C01196=-6.137,-50.981,87.161,174.2492,3.5661,-16836.8641
C01197=-7.391,-55.610,89.719,-178.8088,-0.0035,-16837.5707
C01198=-8.302,-62.896,93.033,-179.1621,0.0008,-16837.5193
C01199=-38.603,-50.345,93.033,179.1623,0.0002,-16867.4799
C01200=-34.096,-44.548,89.719,178.8104,-0.0013,-16867.4296
C01201=-31.710,-40.389,87.161,-174.2479,3.5658,-16868.1360
C01202=-32.743,-37.311,86.112,-176.2272,15.2245,-16871.2692
C01203=-34.176,-35.843,86.067,179.9736,16.5280,-16873.6362
C01204=-35.014,-35.014,86.097,179.9958,16.5019,-16875.0000
C01205=-35.842,-34.176,86.067,-179.9734,16.5280,-16876.3630
C01206=-37.311,-32.743,86.112,176.2272,15.2245,-16878.7308
C01207=-40.389,-31.710,87.161,174.2524,3.5623,-16881.8640
C01208=-44.548,-34.096,89.719,-178.8104,-0.0013,-16882.5704
C01209=-50.345,-38.603,93.033,-179.1623,0.0002,-16882.5201
C01210=-62.896,-8.302,93.033,179.1621,0.0008,-16912.4807
C01211=-55.610,-7.391,89.719,178.8088,-0.0035,-16912.4293
C01212=-50.981,-6.137,87.161,-174.2492,3.5661,-16913.1359
C01213=-49.536,-3.230,86.112,-176.2280,15.2268,-16916.2693
C01214=-49.510,-1.179,86.067,179.9745,16.5281,-16918.6359
C01215=-49.517,0.000,86.097,180.0000,16.4995,-16920.0000
C01216=-49.510,1.178,86.067,-179.9741,16.5281,-16921.3630
C01217=-49.536,3.231,86.112,176.2280,15.2212,-16923.7318
C01218=-50.981,6.137,87.161,174.2492,3.5661,-16926.8641
C01219=-55.610,7.391,89.719,-178.8088,-0.0035,-16927.5707
C01220=-62.896,8.302,93.033,-179.1621,0.0008,-16927.5193
C01221=-50.345,38.603,93.033,179.1623,0.0002,-16957.4799
C01222=-44.548,34.096,89.719,178.8104,-0.0013,-16957.4296
C01223=-40.389,31.710,87.161,-174.2479,3.5658,-16958.1360
C01224=-37.311,32.743,86.112,-176.2272,15.2245,-16961.2692
C01225=-35.843,34.176,86.067,179.9736,16.5280,-16963.6362
C01226=-35.014,35.014,86.097,179.9958,16.5019,-16965.0000
C01227=-34.176,35.842,86.067,-179.9734,16.5280,-16966.3630
C01228=-32.743,37.311,86.112,176.2272,15.2245,-16968.7308
C01229=-31.710,40.389,87.161,174.2524,3.5623,-16971.8640
C01230=-34.096,44.548,89.719,-178.8104,-0.0013,-16972.5704
C01231=-38.603,50.345,93.033,-179.1623,0.0002,-16972.5201
C01232=-8.302,62.896,93.033,179.1621,0.0008,-17002.4807
C01233=-7.391,55.610,89.719,178.8088,-0.0035,-17002.4293
C01234=-6.137,50.981,87.161,-174.2492,3.5661,-17003.1359
C01235=-3.231,49.536,86.112,-176.2280,15.2212,-17006.2682
C01236=-1.178,49.510,86.067,179.9741,16.5281,-17008.6370
C01237=0.000,49.517,86.097,180.0000,16.4995,-17010.0000
C01238=0.000,48.949,88.223,180.0000,13.3790,-17010.0000
C01239=1.127,48.942,88.191,-179.9906,13.4131,-17011.3191
C01240=3.143,48.975,88.238,176.9194,12.2840,-17013.6720
C01241=6.042,50.501,89.306,175.5912,2.6850,-17016.8225
C01242=7.312,55.314,91.898,-179.1905,-0.0028,-17017.5303
C01243=8.270,62.805,95.231,-179.7804,0.0000,-17017.5014
C01244=38.562,50.258,95.231,179.7754,0.0010,-17047.4983
C01245=33.942,44.284,91.898,179.1909,0.0007,-17047.4688
C01246=31.437,39.982,89.306,-175.5900,2.6894,-17048.1772
C01247=32.408,36.853,88.238,-176.9224,12.2833,-17051.3279
C01248=33.811,35.404,88.191,179.9936,13.4108,-17053.6816
C01249=34.612,34.612,88.223,-180.0000,13.3770,-17055.0000
C01250=35.404,33.811,88.191,-179.9936,13.4108,-17056.3184
C01251=36.854,32.408,88.238,176.9223,12.2833,-17058.6728
C01252=39.982,31.437,89.306,175.5945,2.6858,-17061.8228
C01253=44.284,33.942,91.898,-179.1909,0.0007,-17062.5312
C01254=50.258,38.562,95.231,-179.7754,0.0010,-17062.5017
C01255=62.805,8.270,95.231,179.7804,0.0000,-17092.4986
C01256=55.314,7.312,91.898,179.1905,-0.0028,-17092.4697
C01257=50.501,6.042,89.306,-175.5912,2.6850,-17093.1775
C01258=48.975,3.143,88.238,-176.9194,12.2840,-17096.3280
C01259=48.942,1.127,88.191,179.9906,13.4131,-17098.6809
C01260=48.949,0.000,88.223,-180.0000,13.3790,-17100.0000
C01261=48.942,-1.126,88.191,-179.9903,13.4131,-17101.3180
C01262=48.976,-3.143,88.238,176.9195,12.2840,-17103.6719
C01263=50.501,-6.042,89.306,175.5912,2.6850,-17106.8225
C01264=55.314,-7.312,91.898,-179.1905,-0.0028,-17107.5303
C01265=62.805,-8.270,95.231,-179.7804,0.0000,-17107.5014
C01266=50.258,-38.562,95.231,179.7754,0.0010,-17137.4983
C01267=44.284,-33.942,91.898,179.1909,0.0007,-17137.4688
C01268=39.982,-31.437,89.306,-175.5900,2.6894,-17138.1772
C01269=36.853,-32.408,88.238,-176.9224,12.2833,-17141.3279
C01270=35.404,-33.811,88.191,179.9936,13.4108,-17143.6816
C01271=34.612,-34.612,88.223,-180.0000,13.3770,-17145.0000
C01272=33.811,-35.404,88.191,-179.9936,13.4108,-17146.3184
C01273=32.408,-36.854,88.238,176.9223,12.2833,-17148.6728
C01274=31.437,-39.982,89.306,175.5945,2.6858,-17151.8228
C01275=33.942,-44.284,91.898,-179.1909,0.0007,-17152.5312
C01276=38.562,-50.258,95.231,-179.7754,0.0010,-17152.5017
C01277=8.270,-62.805,95.231,179.7804,0.0000,-17182.4986
C01278=7.312,-55.314,91.898,179.1905,-0.0028,-17182.4697
C01279=6.042,-50.501,89.306,-175.5912,2.6850,-17183.1775
C01280=3.143,-48.975,88.238,-176.9194,12.2840,-17186.3280
C01281=1.127,-48.942,88.191,179.9906,13.4131,-17188.6809
C01282=0.000,-48.949,88.223,-180.0000,13.3790,-17190.0000
C01283=0.000,-48.949,88.223,-180.0000,13.3790,-17190.0000
C01284=-1.126,-48.942,88.191,-179.9903,13.4131,-17191.3180
C01285=-3.143,-48.976,88.238,176.9195,12.2840,-17193.6719
C01286=-6.042,-50.501,89.306,175.5912,2.6850,-17196.8225
C01287=-7.312,-55.314,91.898,-179.1905,-0.0028,-17197.5303
C01288=-8.270,-62.805,95.231,-179.7804,0.0000,-17197.5014
C01289=-38.562,-50.258,95.231,179.7754,0.0010,-17227.4983
C01290=-33.942,-44.284,91.898,179.1909,0.0007,-17227.4688
C01291=-31.437,-39.982,89.306,-175.5900,2.6894,-17228.1772
C01292=-32.408,-36.853,88.238,-176.9224,12.2833,-17231.3279
C01293=-33.811,-35.404,88.191,179.9936,13.4108,-17233.6816
C01294=-34.612,-34.612,88.223,180.0000,13.3770,-17235.0000
C01295=-35.404,-33.811,88.191,-179.9936,13.4108,-17236.3184
C01296=-36.854,-32.408,88.238,176.9223,12.2833,-17238.6728
C01297=-39.982,-31.437,89.306,175.5945,2.6858,-17241.8228
C01298=-44.284,-33.942,91.898,-179.1909,0.0007,-17242.5312
C01299=-50.258,-38.562,95.231,-179.7754,0.0010,-17242.5017
C01300=-62.805,-8.270,95.231,179.7804,0.0000,-17272.4986
C01301=-55.314,-7.312,91.898,179.1905,-0.0028,-17272.4697
C01302=-50.501,-6.042,89.306,-175.5912,2.6850,-17273.1775
C01303=-48.975,-3.143,88.238,-176.9194,12.2840,-17276.3280
C01304=-48.942,-1.127,88.191,179.9906,13.4131,-17278.6809
C01305=-48.949,0.000,88.223,-180.0000,13.3790,-17280.0000
C01306=-48.942,1.126,88.191,-179.9903,13.4131,-17281.3180
C01307=-48.976,3.143,88.238,176.9195,12.2840,-17283.6719
C01308=-50.501,6.042,89.306,175.5912,2.6850,-17286.8225
C01309=-55.314,7.312,91.898,-179.1905,-0.0028,-17287.5303
C01310=-62.805,8.270,95.231,-179.7804,0.0000,-17287.5014
C01311=-50.258,38.562,95.231,179.7754,0.0010,-17317.4983
C01312=-44.284,33.942,91.898,179.1909,0.0007,-17317.4688
C01313=-39.982,31.437,89.306,-175.5900,2.6894,-17318.1772
C01314=-36.853,32.408,88.238,-176.9224,12.2833,-17321.3279
C01315=-35.404,33.811,88.191,179.9936,13.4108,-17323.6816
C01316=-34.612,34.612,88.223,180.0000,13.3770,-17325.0000
C01317=-33.811,35.404,88.191,-179.9936,13.4108,-17326.3184
C01318=-32.408,36.854,88.238,176.9223,12.2833,-17328.6728
C01319=-31.437,39.982,89.306,175.5945,2.6858,-17331.8228
C01320=-33.942,44.284,91.898,-179.1909,0.0007,-17332.5312
C01321=-38.562,50.258,95.231,-179.7754,0.0010,-17332.5017
C01322=-8.270,62.805,95.231,179.7804,0.0000,-17362.4986
C01323=-7.312,55.314,91.898,179.1905,-0.0028,-17362.4697
C01324=-6.042,50.501,89.306,-175.5912,2.6850,-17363.1775
C01325=-3.143,48.976,88.238,-176.9195,12.2840,-17366.3281
C01326=-1.126,48.942,88.191,179.9903,13.4131,-17368.6820
C01327=0.000,48.949,88.223,-180.0000,13.3790,-17370.0000
C01328=0.000,48.503,90.377,-180.0000,9.9625,-17370.0000
C01329=1.086,48.496,90.345,-179.9994,10.0055,-17371.2828
C01330=3.075,48.536,90.393,177.6967,9.1102,-17373.6251
C01331=5.972,50.143,91.476,176.9766,1.8184,-17376.7919
C01332=7.266,55.138,94.090,-179.6070,-0.0002,-17377.5071
C01333=33.851,44.126,94.090,179.6115,-0.0019,-17407.4934
C01334=31.234,39.679,91.476,-176.9779,1.8180,-17408.2087
C01335=32.146,36.494,90.393,-177.6994,9.1088,-17411.3754
C01336=33.524,35.059,90.345,-179.9960,10.0034,-17413.7178
C01337=34.297,34.297,90.377,180.0000,9.9681,-17415.0000
C01338=35.059,33.525,90.345,179.9962,10.0034,-17416.2813
C01339=36.495,32.146,90.393,177.6954,9.1045,-17418.6253
C01340=39.679,31.234,91.476,176.9779,1.8180,-17421.7913
C01341=44.126,33.851,94.090,-179.6115,-0.0019,-17422.5066
C01342=55.138,7.266,94.090,179.6070,-0.0002,-17452.4929
C01343=50.143,5.972,91.476,-176.9766,1.8184,-17453.2081
C01344=48.536,3.075,90.393,-177.6967,9.1102,-17456.3749
C01345=48.496,1.086,90.345,179.9994,10.0055,-17458.7172
C01346=48.503,0.000,90.377,-180.0000,9.9625,-17460.0000
C01347=48.496,-1.085,90.345,-179.9992,10.0055,-17461.2817
C01348=48.536,-3.075,90.393,177.6967,9.1102,-17463.6251
C01349=50.143,-5.972,91.476,176.9766,1.8184,-17466.7919
C01350=55.138,-7.266,94.090,-179.6070,-0.0002,-17467.5071
C01351=44.126,-33.851,94.090,179.6115,-0.0019,-17497.4934
C01352=39.679,-31.234,91.476,-176.9779,1.8180,-17498.2087
C01353=36.494,-32.146,90.393,-177.6994,9.1088,-17501.3754
C01354=35.059,-33.524,90.345,-179.9960,10.0034,-17503.7178
C01355=34.297,-34.297,90.377,180.0000,9.9681,-17505.0000
C01356=33.525,-35.059,90.345,179.9962,10.0034,-17506.2813
C01357=32.146,-36.495,90.393,177.6954,9.1045,-17508.6253
C01358=31.234,-39.679,91.476,176.9779,1.8180,-17511.7913
C01359=33.851,-44.126,94.090,-179.6115,-0.0019,-17512.5066
C01360=7.266,-55.138,94.090,179.6070,-0.0002,-17542.4929
C01361=5.972,-50.143,91.476,-176.9766,1.8184,-17543.2081
C01362=3.075,-48.536,90.393,-177.6967,9.1102,-17546.3749
C01363=1.086,-48.496,90.345,179.9994,10.0055,-17548.7172
C01364=0.000,-48.503,90.377,-180.0000,9.9625,-17550.0000
C01365=0.000,-48.503,90.377,-180.0000,9.9625,-17550.0000
C01366=-1.085,-48.496,90.345,-179.9992,10.0055,-17551.2817
C01367=-3.075,-48.536,90.393,177.6967,9.1102,-17553.6251
C01368=-5.972,-50.143,91.476,176.9766,1.8184,-17556.7919
C01369=-7.266,-55.138,94.090,-179.6070,-0.0002,-17557.5071
C01370=-33.851,-44.126,94.090,179.6115,-0.0019,-17587.4934
C01371=-31.234,-39.679,91.476,-176.9779,1.8180,-17588.2087
C01372=-32.146,-36.494,90.393,-177.6994,9.1088,-17591.3754
C01373=-33.524,-35.059,90.345,-179.9960,10.0034,-17593.7178
C01374=-34.297,-34.297,90.377,-180.0000,9.9681,-17595.0000
C01375=-35.059,-33.525,90.345,179.9962,10.0034,-17596.2813
C01376=-36.495,-32.146,90.393,177.6954,9.1045,-17598.6253
C01377=-39.679,-31.234,91.476,176.9779,1.8180,-17601.7913
C01378=-44.126,-33.851,94.090,-179.6115,-0.0019,-17602.5066
C01379=-55.138,-7.266,94.090,179.6070,-0.0002,-17632.4929
C01380=-50.143,-5.972,91.476,-176.9766,1.8184,-17633.2081
C01381=-48.536,-3.075,90.393,-177.6967,9.1102,-17636.3749
C01382=-48.496,-1.086,90.345,179.9994,10.0055,-17638.7172
C01383=-48.503,0.000,90.377,-180.0000,9.9625,-17640.0000
C01384=-48.496,1.085,90.345,-179.9992,10.0055,-17641.2817
C01385=-48.536,3.075,90.393,177.6967,9.1102,-17643.6251
C01386=-50.143,5.972,91.476,176.9766,1.8184,-17646.7919
C01387=-55.138,7.266,94.090,-179.6070,-0.0002,-17647.5071
C01388=-44.126,33.851,94.090,179.6115,-0.0019,-17677.4934
C01389=-39.679,31.234,91.476,-176.9779,1.8180,-17678.2087
C01390=-36.494,32.146,90.393,-177.6994,9.1088,-17681.3754
C01391=-35.059,33.524,90.345,-179.9960,10.0034,-17683.7178
C01392=-34.297,34.297,90.377,-180.0000,9.9681,-17685.0000
C01393=-33.525,35.059,90.345,179.9962,10.0034,-17686.2813
C01394=-32.146,36.495,90.393,177.6954,9.1045,-17688.6253
C01395=-31.234,39.679,91.476,176.9779,1.8180,-17691.7913
C01396=-33.851,44.126,94.090,-179.6115,-0.0019,-17692.5066
C01397=-7.266,55.138,94.090,179.6070,-0.0002,-17722.4929
C01398=-5.972,50.143,91.476,-176.9766,1.8184,-17723.2081
C01399=-3.075,48.536,90.393,-177.6967,9.1102,-17726.3749
C01400=-1.085,48.496,90.345,179.9992,10.0055,-17728.7183
C01401=0.000,48.503,90.377,180.0000,9.9625,-17730.0000
C01402=0.000,48.191,92.555,180.0000,6.2750,-17730.0000
C01403=1.057,48.183,92.523,179.9934,6.3226,-17731.2567
C01404=3.027,48.229,92.571,178.5501,5.7076,-17733.5913
C01405=5.927,49.917,93.664,178.4157,0.9490,-17736.7714
C01406=31.106,39.488,93.664,-178.4140,0.9504,-17768.2287
C01407=31.963,36.244,92.571,-178.5471,5.7094,-17771.4086
C01408=33.323,34.818,92.523,-179.9953,6.3224,-17773.7431
C01409=34.076,34.076,92.555,-180.0000,6.2761,-17775.0000
C01410=34.818,33.324,92.523,179.9954,6.3224,-17776.2560
C01411=36.244,31.963,92.571,178.5471,5.7094,-17778.5914
C01412=39.488,31.106,93.664,178.4140,0.9504,-17781.7713
C01413=49.917,5.927,93.664,-178.4157,0.9490,-17813.2286
C01414=48.229,3.027,92.571,-178.5501,5.7076,-17816.4087
C01415=48.183,1.057,92.523,-179.9934,6.3226,-17818.7433
C01416=48.191,0.000,92.555,180.0000,6.2750,-17820.0000
C01417=48.183,-1.057,92.523,179.9934,6.3226,-17821.2567
C01418=48.229,-3.027,92.571,178.5443,5.7073,-17823.5913
C01419=49.918,-5.927,93.664,178.4157,0.9490,-17826.7713
C01420=39.488,-31.106,93.664,-178.4140,0.9504,-17858.2287
C01421=36.244,-31.963,92.571,-178.5471,5.7094,-17861.4086
C01422=34.818,-33.323,92.523,-179.9953,6.3224,-17863.7431
C01423=34.076,-34.076,92.555,-180.0000,6.2761,-17865.0000
C01424=33.324,-34.818,92.523,179.9954,6.3224,-17866.2560
C01425=31.963,-36.244,92.571,178.5471,5.7094,-17868.5914
C01426=31.106,-39.488,93.664,178.4140,0.9504,-17871.7713
C01427=5.927,-49.917,93.664,-178.4157,0.9490,-17903.2286
C01428=3.027,-48.229,92.571,-178.5501,5.7076,-17906.4087
C01429=1.057,-48.183,92.523,-179.9934,6.3226,-17908.7433
C01430=0.000,-48.191,92.555,180.0000,6.2750,-17910.0000
C01431=0.000,-48.191,92.555,180.0000,6.2750,-17910.0000
C01432=-1.057,-48.183,92.523,179.9934,6.3226,-17911.2567
C01433=-3.027,-48.229,92.571,178.5443,5.7073,-17913.5913
C01434=-5.927,-49.918,93.664,178.4157,0.9490,-17916.7713
C01435=-31.106,-39.488,93.664,-178.4140,0.9504,-17948.2287
C01436=-31.963,-36.244,92.571,-178.5471,5.7094,-17951.4086
C01437=-33.323,-34.818,92.523,-179.9953,6.3224,-17953.7431
C01438=-34.076,-34.076,92.555,-180.0000,6.2761,-17955.0000
C01439=-34.818,-33.324,92.523,179.9954,6.3224,-17956.2560
C01440=-36.244,-31.963,92.571,178.5471,5.7094,-17958.5914
C01441=-39.488,-31.106,93.664,178.4140,0.9504,-17961.7713
C01442=-49.917,-5.927,93.664,-178.4157,0.9490,-17993.2286
C01443=-48.229,-3.027,92.571,-178.5501,5.7076,-17996.4087
C01444=-48.183,-1.057,92.523,-179.9934,6.3226,-17998.7433
C01445=-48.191,0.000,92.555,180.0000,6.2750,-18000.0000
C01446=-48.183,1.057,92.523,179.9934,6.3226,-18001.2567
C01447=-48.229,3.027,92.571,178.5443,5.7073,-18003.5913
C01448=-49.918,5.927,93.664,178.4157,0.9490,-18006.7713
C01449=-39.488,31.106,93.664,-178.4140,0.9504,-18038.2287
C01450=-36.244,31.963,92.571,-178.5471,5.7094,-18041.4086
C01451=-34.818,33.323,92.523,-179.9953,6.3224,-18043.7431
C01452=-34.076,34.076,92.555,-180.0000,6.2761,-18045.0000
C01453=-33.324,34.818,92.523,179.9954,6.3224,-18046.2560
C01454=-31.963,36.244,92.571,178.5471,5.7094,-18048.5914
C01455=-31.106,39.488,93.664,178.4140,0.9504,-18051.7713
C01456=-5.927,49.918,93.664,-178.4157,0.9490,-18083.2287
C01457=-3.027,48.229,92.571,-178.5443,5.7073,-18086.4087
C01458=-1.057,48.183,92.523,-179.9934,6.3226,-18088.7433
C01459=0.000,48.191,92.555,-180.0000,6.2750,-18090.0000
C01460=0.000,48.026,94.749,-180.0000,2.3325,-18090.0000
C01461=1.042,48.016,94.716,179.9997,2.3906,-18091.2432
C01462=3.002,48.067,94.764,179.4608,2.1024,-18093.5737
C01463=5.911,49.834,95.862,179.9066,0.0582,-18096.7645
C01464=31.058,39.418,95.862,-179.9039,0.0539,-18128.2351
C01465=31.866,36.111,94.764,-179.4625,2.1022,-18131.4267
C01466=33.216,34.689,94.716,-179.9968,2.3916,-18133.7573
C01467=33.959,33.959,94.749,180.0000,2.3342,-18135.0000
C01468=34.689,33.216,94.716,179.9968,2.3916,-18136.2427
C01469=36.111,31.865,94.764,179.4624,2.1022,-18138.5742
C01470=39.418,31.058,95.862,179.9039,0.0539,-18141.7649
C01471=49.834,5.911,95.862,-179.9066,0.0582,-18173.2355
C01472=48.067,3.002,94.764,-179.4608,2.1024,-18176.4263
C01473=48.016,1.042,94.716,-179.9997,2.3906,-18178.7568
C01474=48.026,0.000,94.749,-180.0000,2.3325,-18180.0000
C01475=48.016,-1.041,94.716,179.9998,2.3906,-18181.2420
C01476=48.067,-3.002,94.764,179.4608,2.1024,-18183.5737
C01477=49.834,-5.911,95.862,179.9066,0.0582,-18186.7645
C01478=39.418,-31.058,95.862,-179.9039,0.0539,-18218.2351
C01479=36.111,-31.866,94.764,-179.4625,2.1022,-18221.4267
C01480=34.689,-33.216,94.716,-179.9968,2.3916,-18223.7573
C01481=33.959,-33.959,94.749,180.0000,2.3342,-18225.0000
C01482=33.216,-34.689,94.716,179.9968,2.3916,-18226.2427
C01483=31.865,-36.111,94.764,179.4624,2.1022,-18228.5742
C01484=31.058,-39.418,95.862,179.9039,0.0539,-18231.7649
C01485=5.911,-49.834,95.862,-179.9066,0.0582,-18263.2355
C01486=3.002,-48.067,94.764,-179.4608,2.1024,-18266.4263
C01487=1.042,-48.016,94.716,-179.9997,2.3906,-18268.7568
C01488=0.000,-48.026,94.749,-180.0000,2.3325,-18270.0000
C01489=0.000,-48.026,94.749,-180.0000,2.3325,-18270.0000
C01490=-1.041,-48.016,94.716,179.9998,2.3906,-18271.2420
C01491=-3.002,-48.067,94.764,179.4608,2.1024,-18273.5737
C01492=-5.911,-49.834,95.862,179.9066,0.0582,-18276.7645
C01493=-31.058,-39.418,95.862,-179.9039,0.0539,-18308.2351
C01494=-31.866,-36.111,94.764,-179.4625,2.1022,-18311.4267
C01495=-33.216,-34.689,94.716,-179.9968,2.3916,-18313.7573
C01496=-33.959,-33.959,94.749,180.0000,2.3342,-18315.0000
C01497=-34.689,-33.216,94.716,179.9968,2.3916,-18316.2427
C01498=-36.111,-31.865,94.764,179.4624,2.1022,-18318.5742
C01499=-39.418,-31.058,95.862,179.9039,0.0539,-18321.7649
C01500=-49.834,-5.911,95.862,-179.9066,0.0582,-18353.2355
C01501=-48.067,-3.002,94.764,-179.4608,2.1024,-18356.4263
C01502=-48.016,-1.042,94.716,-179.9997,2.3906,-18358.7568
C01503=-48.026,0.000,94.749,-180.0000,2.3325,-18360.0000
C01504=-48.016,1.041,94.716,179.9998,2.3906,-18361.2420
C01505=-48.067,3.002,94.764,179.4608,2.1024,-18363.5737
C01506=-49.834,5.911,95.862,179.9066,0.0582,-18366.7645
C01507=-39.418,31.058,95.862,-179.9039,0.0539,-18398.2351
C01508=-36.111,31.866,94.764,-179.4625,2.1022,-18401.4267
C01509=-34.689,33.216,94.716,-179.9968,2.3916,-18403.7573
C01510=-33.959,33.959,94.749,180.0000,2.3342,-18405.0000
C01511=-33.216,34.689,94.716,179.9968,2.3916,-18406.2427
C01512=-31.865,36.111,94.764,179.4624,2.1022,-18408.5742
C01513=-31.058,39.418,95.862,179.9039,0.0539,-18411.7649
C01514=-5.911,49.834,95.862,-179.9066,0.0582,-18443.2355
C01515=-3.002,48.067,94.764,-179.4608,2.1024,-18446.4263
C01516=-1.041,48.016,94.716,-179.9998,2.3906,-18448.7580
C01517=0.000,48.026,94.749,-180.0000,2.3325,-18450.0000
///TOOL 0
///POSTYPE ANGLE
///ANGLE
EC00000=0.0000,14346.8537
EC00001=0.0000,14347.6887
EC00002=0.0000,14350.6829
EC00003=0.0000,14353.1899
EC00004=0.0000,14355.0000
EC00005=0.0000,14356.8101
EC00006=0.0000,14359.3178
EC00007=0.0000,14362.3119
EC00008=0.0000,14363.1463
EC00009=0.0000,14363.1205
EC00010=0.0000,14362.9934
EC00011=0.0000,14362.8957
EC00012=0.0000,14362.9735
EC00013=0.0000,14364.6500
EC00014=0.0000,14367.6087
EC00015=0.0000,14371.3401
EC00016=0.0000,14375.4161
EC00017=0.0000,14379.5839
EC00018=0.0000,14383.6602
EC00019=0.0000,14387.3912
EC00020=0.0000,14390.3496
EC00021=0.0000,14392.0267
EC00022=0.0000,14392.1045
EC00023=0.0000,14392.0068
EC00024=0.0000,14391.8791
EC00025=0.0000,14391.8541
EC00026=0.0000,14392.6890
EC00027=0.0000,14395.6832
EC00028=0.0000,14398.1896
EC00029=0.0000,14400.0000
EC00030=0.0000,14401.8094
EC00031=0.0000,14404.3178
EC00032=0.0000,14407.3110
EC00033=0.0000,14408.1459
EC00034=0.0000,14408.1209
EC00035=0.0000,14407.9932
EC00036=0.0000,14407.8955
EC00037=0.0000,14407.9733
EC00038=0.0000,14409.6504
EC00039=0.0000,14412.6088
EC00040=0.0000,14416.3398
EC00041=0.0000,14420.4161
EC00042=0.0000,14424.5839
EC00043=0.0000,14428.6599
EC00044=0.0000,14432.3913
EC00045=0.0000,14435.3500
EC00046=0.0000,14437.0265
EC00047=0.0000,14437.1043
EC00048=0.0000,14437.0066
EC00049=0.0000,14436.8795
EC00050=0.0000,14436.8537
EC00051=0.0000,14437.6887
EC00052=0.0000,14440.6829
EC00053=0.0000,14443.1899
EC00054=0.0000,14445.0000
EC00055=0.0000,14446.8101
EC00056=0.0000,14449.3178
EC00057=0.0000,14452.3119
EC00058=0.0000,14453.1463
EC00059=0.0000,14453.1205
EC00060=0.0000,14452.9934
EC00061=0.0000,14452.8957
EC00062=0.0000,14452.9735
EC00063=0.0000,14454.6500
EC00064=0.0000,14457.6087
EC00065=0.0000,14461.3401
EC00066=0.0000,14465.4161
EC00067=0.0000,14469.5839
EC00068=0.0000,14473.6602
EC00069=0.0000,14477.3912
EC00070=0.0000,14480.3496
EC00071=0.0000,14482.0267
EC00072=0.0000,14482.1045
EC00073=0.0000,14482.0068
EC00074=0.0000,14481.8791
EC00075=0.0000,14481.8541
EC00076=0.0000,14482.6890
EC00077=0.0000,14485.6822
EC00078=0.0000,14488.1906
EC00079=0.0000,14490.0000
EC00080=0.0000,14490.0000
EC00081=0.0000,14491.7406
EC00082=0.0000,14494.2255
EC00083=0.0000,14497.2387
EC00084=0.0000,14498.0440
EC00085=0.0000,14497.9981
EC00086=0.0000,14497.8709
EC00087=0.0000,14497.7793
EC00088=0.0000,14497.8555
EC00089=0.0000,14499.5452
EC00090=0.0000,14502.5282
EC00091=0.0000,14506.2898
EC00092=0.0000,14510.3994
EC00093=0.0000,14514.6009
EC00094=0.0000,14518.7101
EC00095=0.0000,14522.4718
EC00096=0.0000,14525.4547
EC00097=0.0000,14527.1446
EC00098=0.0000,14527.2208
EC00099=0.0000,14527.1290
EC00100=0.0000,14527.0022
EC00101=0.0000,14526.9563
EC00102=0.0000,14527.7605
EC00103=0.0000,14530.7744
EC00104=0.0000,14533.2595
EC00105=0.0000,14535.0000
EC00106=0.0000,14536.7398
EC00107=0.0000,14539.2256
EC00108=0.0000,14542.2395
EC00109=0.0000,14543.0437
EC00110=0.0000,14542.9978
EC00111=0.0000,14542.8710
EC00112=0.0000,14542.7792
EC00113=0.0000,14542.8554
EC00114=0.0000,14544.5453
EC00115=0.0000,14547.5282
EC00116=0.0000,14551.2899
EC00117=0.0000,14555.3991
EC00118=0.0000,14559.6006
EC00119=0.0000,14563.7102
EC00120=0.0000,14567.4718
EC00121=0.0000,14570.4548
EC00122=0.0000,14572.1445
EC00123=0.0000,14572.2207
EC00124=0.0000,14572.1291
EC00125=0.0000,14572.0019
EC00126=0.0000,14571.9560
EC00127=0.0000,14572.7613
EC00128=0.0000,14575.7745
EC00129=0.0000,14578.2594
EC00130=0.0000,14580.0000
EC00131=0.0000,14581.7396
EC00132=0.0000,14584.2255
EC00133=0.0000,14587.2387
EC00134=0.0000,14588.0440
EC00135=0.0000,14587.9981
EC00136=0.0000,14587.8709
EC00137=0.0000,14587.7793
EC00138=0.0000,14587.8555
EC00139=0.0000,14589.5452
EC00140=0.0000,14592.5282
EC00141=0.0000,14596.2898
EC00142=0.0000,14600.3994
EC00143=0.0000,14604.6009
EC00144=0.0000,14608.7101
EC00145=0.0000,14612.4718
EC00146=0.0000,14615.4547
EC00147=0.0000,14617.1446
EC00148=0.0000,14617.2208
EC00149=0.0000,14617.1290
EC00150=0.0000,14617.0022
EC00151=0.0000,14616.9563
EC00152=0.0000,14617.7605
EC00153=0.0000,14620.7744
EC00154=0.0000,14623.2595
EC00155=0.0000,14625.0000
EC00156=0.0000,14626.7398
EC00157=0.0000,14629.2256
EC00158=0.0000,14632.2395
EC00159=0.0000,14633.0437
EC00160=0.0000,14632.9978
EC00161=0.0000,14632.8710
EC00162=0.0000,14632.7792
EC00163=0.0000,14632.8554
EC00164=0.0000,14634.5453
EC00165=0.0000,14637.5282
EC00166=0.0000,14641.2899
EC00167=0.0000,14645.3991
EC00168=0.0000,14649.6006
EC00169=0.0000,14653.7102
EC00170=0.0000,14657.4718
EC00171=0.0000,14660.4548
EC00172=0.0000,14662.1445
EC00173=0.0000,14662.2207
EC00174=0.0000,14662.1291
EC00175=0.0000,14662.0019
EC00176=0.0000,14661.9560
EC00177=0.0000,14662.7613
EC00178=0.0000,14665.7745
EC00179=0.0000,14668.2594
EC00180=0.0000,14670.0000
EC00181=0.0000,14670.0000
EC00182=0.0000,14671.7396
EC00183=0.0000,14674.2255
EC00184=0.0000,14677.2387
EC00185=0.0000,14678.0440
EC00186=0.0000,14677.9981
EC00187=0.0000,14677.8709
EC00188=0.0000,14677.7793
EC00189=0.0000,14677.8555
EC00190=0.0000,14679.5452
EC00191=0.0000,14682.5282
EC00192=0.0000,14686.2898
EC00193=0.0000,14690.3994
EC00194=0.0000,14694.6009
EC00195=0.0000,14698.7101
EC00196=0.0000,14702.4718
EC00197=0.0000,14705.4547
EC00198=0.0000,14707.1446
EC00199=0.0000,14707.2208
EC00200=0.0000,14707.1290
EC00201=0.0000,14707.0022
EC00202=0.0000,14706.9563
EC00203=0.0000,14707.7605
EC00204=0.0000,14710.7744
EC00205=0.0000,14713.2595
EC00206=0.0000,14715.0000
EC00207=0.0000,14716.7398
EC00208=0.0000,14719.2256
EC00209=0.0000,14722.2395
EC00210=0.0000,14723.0437
EC00211=0.0000,14722.9978
EC00212=0.0000,14722.8710
EC00213=0.0000,14722.7792
EC00214=0.0000,14722.8554
EC00215=0.0000,14724.5453
EC00216=0.0000,14727.5282
EC00217=0.0000,14731.2899
EC00218=0.0000,14735.3991
EC00219=0.0000,14739.6006
EC00220=0.0000,14743.7102
EC00221=0.0000,14747.4718
EC00222=0.0000,14750.4548
EC00223=0.0000,14752.1445
EC00224=0.0000,14752.2207
EC00225=0.0000,14752.1291
EC00226=0.0000,14752.0019
EC00227=0.0000,14751.9560
EC00228=0.0000,14752.7613
EC00229=0.0000,14755.7745
EC00230=0.0000,14758.2594
EC00231=0.0000,14760.0000
EC00232=0.0000,14761.7396
EC00233=0.0000,14764.2255
EC00234=0.0000,14767.2387
EC00235=0.0000,14768.0440
EC00236=0.0000,14767.9981
EC00237=0.0000,14767.8709
EC00238=0.0000,14767.7793
EC00239=0.0000,14767.8555
EC00240=0.0000,14769.5452
EC00241=0.0000,14772.5282
EC00242=0.0000,14776.2898
EC00243=0.0000,14780.3994
EC00244=0.0000,14784.6009
EC00245=0.0000,14788.7101
EC00246=0.0000,14792.4718
EC00247=0.0000,14795.4547
EC00248=0.0000,14797.1446
EC00249=0.0000,14797.2208
EC00250=0.0000,14797.1290
EC00251=0.0000,14797.0022
EC00252=0.0000,14796.9563
EC00253=0.0000,14797.7605
EC00254=0.0000,14800.7744
EC00255=0.0000,14803.2595
EC00256=0.0000,14805.0000
EC00257=0.0000,14806.7398
EC00258=0.0000,14809.2256
EC00259=0.0000,14812.2395
EC00260=0.0000,14813.0437
EC00261=0.0000,14812.9978
EC00262=0.0000,14812.8710
EC00263=0.0000,14812.7792
EC00264=0.0000,14812.8554
EC00265=0.0000,14814.5453
EC00266=0.0000,14817.5282
EC00267=0.0000,14821.2899
EC00268=0.0000,14825.3991
EC00269=0.0000,14829.6006
EC00270=0.0000,14833.7102
EC00271=0.0000,14837.4718
EC00272=0.0000,14840.4548
EC00273=0.0000,14842.1445
EC00274=0.0000,14842.2207
EC00275=0.0000,14842.1291
EC00276=0.0000,14842.0019
EC00277=0.0000,14841.9560
EC00278=0.0000,14842.7613
EC00279=0.0000,14845.7745
EC00280=0.0000,14848.2604
EC00281=0.0000,14850.0000
EC00282=0.0000,14850.0000
EC00283=0.0000,14851.6706
EC00284=0.0000,14854.1339
EC00285=0.0000,14857.1680
EC00286=0.0000,14857.9465
EC00287=0.0000,14857.8844
EC00288=0.0000,14857.7630
EC00289=0.0000,14857.6803
EC00290=0.0000,14857.7585
EC00291=0.0000,14859.4604
EC00292=0.0000,14862.4636
EC00293=0.0000,14866.2505
EC00294=0.0000,14870.3860
EC00295=0.0000,14874.6140
EC00296=0.0000,14878.7498
EC00297=0.0000,14882.5363
EC00298=0.0000,14885.5394
EC00299=0.0000,14887.2413
EC00300=0.0000,14887.3191
EC00301=0.0000,14887.2369
EC00302=0.0000,14887.1159
EC00303=0.0000,14887.0536
EC00304=0.0000,14887.8325
EC00305=0.0000,14890.8660
EC00306=0.0000,14893.3290
EC00307=0.0000,14895.0000
EC00308=0.0000,14896.6710
EC00309=0.0000,14899.1340
EC00310=0.0000,14902.1675
EC00311=0.0000,14902.9464
EC00312=0.0000,14902.8841
EC00313=0.0000,14902.7631
EC00314=0.0000,14902.6809
EC00315=0.0000,14902.7587
EC00316=0.0000,14904.4606
EC00317=0.0000,14907.4637
EC00318=0.0000,14911.2502
EC00319=0.0000,14915.3860
EC00320=0.0000,14919.6140
EC00321=0.0000,14923.7495
EC00322=0.0000,14927.5364
EC00323=0.0000,14930.5396
EC00324=0.0000,14932.2415
EC00325=0.0000,14932.3197
EC00326=0.0000,14932.2370
EC00327=0.0000,14932.1156
EC00328=0.0000,14932.0535
EC00329=0.0000,14932.8320
EC00330=0.0000,14935.8661
EC00331=0.0000,14938.3294
EC00332=0.0000,14940.0000
EC00333=0.0000,14941.6706
EC00334=0.0000,14944.1349
EC00335=0.0000,14947.1678
EC00336=0.0000,14947.9465
EC00337=0.0000,14947.8844
EC00338=0.0000,14947.7630
EC00339=0.0000,14947.6803
EC00340=0.0000,14947.7585
EC00341=0.0000,14949.4604
EC00342=0.0000,14952.4636
EC00343=0.0000,14956.2505
EC00344=0.0000,14960.3860
EC00345=0.0000,14964.6140
EC00346=0.0000,14968.7498
EC00347=0.0000,14972.5363
EC00348=0.0000,14975.5394
EC00349=0.0000,14977.2413
EC00350=0.0000,14977.3191
EC00351=0.0000,14977.2369
EC00352=0.0000,14977.1159
EC00353=0.0000,14977.0536
EC00354=0.0000,14977.8325
EC00355=0.0000,14980.8660
EC00356=0.0000,14983.3290
EC00357=0.0000,14985.0000
EC00358=0.0000,14986.6710
EC00359=0.0000,14989.1340
EC00360=0.0000,14992.1675
EC00361=0.0000,14992.9464
EC00362=0.0000,14992.8841
EC00363=0.0000,14992.7631
EC00364=0.0000,14992.6809
EC00365=0.0000,14992.7587
EC00366=0.0000,14994.4606
EC00367=0.0000,14997.4637
EC00368=0.0000,15001.2502
EC00369=0.0000,15005.3860
EC00370=0.0000,15009.6140
EC00371=0.0000,15013.7495
EC00372=0.0000,15017.5364
EC00373=0.0000,15020.5396
EC00374=0.0000,15022.2415
EC00375=0.0000,15022.3197
EC00376=0.0000,15022.2370
EC00377=0.0000,15022.1156
EC00378=0.0000,15022.0535
EC00379=0.0000,15022.8320
EC00380=0.0000,15025.8661
EC00381=0.0000,15028.3294
EC00382=0.0000,15030.0000
EC00383=0.0000,15030.0000
EC00384=0.0000,15031.6706
EC00385=0.0000,15034.1349
EC00386=0.0000,15037.1678
EC00387=0.0000,15037.9465
EC00388=0.0000,15037.8844
EC00389=0.0000,15037.7630
EC00390=0.0000,15037.6803
EC00391=0.0000,15037.7585
EC00392=0.0000,15039.4604
EC00393=0.0000,15042.4636
EC00394=0.0000,15046.2505
EC00395=0.0000,15050.3860
EC00396=0.0000,15054.6140
EC00397=0.0000,15058.7498
EC00398=0.0000,15062.5363
EC00399=0.0000,15065.5394
EC00400=0.0000,15067.2413
EC00401=0.0000,15067.3191
EC00402=0.0000,15067.2369
EC00403=0.0000,15067.1159
EC00404=0.0000,15067.0536
EC00405=0.0000,15067.8325
EC00406=0.0000,15070.8660
EC00407=0.0000,15073.3290
EC00408=0.0000,15075.0000
EC00409=0.0000,15076.6710
EC00410=0.0000,15079.1340
EC00411=0.0000,15082.1675
EC00412=0.0000,15082.9464
EC00413=0.0000,15082.8841
EC00414=0.0000,15082.7631
EC00415=0.0000,15082.6809
EC00416=0.0000,15082.7587
EC00417=0.0000,15084.4606
EC00418=0.0000,15087.4637
EC00419=0.0000,15091.2502
EC00420=0.0000,15095.3860
EC00421=0.0000,15099.6140
EC00422=0.0000,15103.7495
EC00423=0.0000,15107.5364
EC00424=0.0000,15110.5396
EC00425=0.0000,15112.2415
EC00426=0.0000,15112.3197
EC00427=0.0000,15112.2370
EC00428=0.0000,15112.1156
EC00429=0.0000,15112.0535
EC00430=0.0000,15112.8320
EC00431=0.0000,15115.8661
EC00432=0.0000,15118.3294
EC00433=0.0000,15120.0000
EC00434=0.0000,15121.6706
EC00435=0.0000,15124.1349
EC00436=0.0000,15127.1678
EC00437=0.0000,15127.9465
EC00438=0.0000,15127.8844
EC00439=0.0000,15127.7630
EC00440=0.0000,15127.6803
EC00441=0.0000,15127.7585
EC00442=0.0000,15129.4604
EC00443=0.0000,15132.4636
EC00444=0.0000,15136.2505
EC00445=0.0000,15140.3860
EC00446=0.0000,15144.6140
